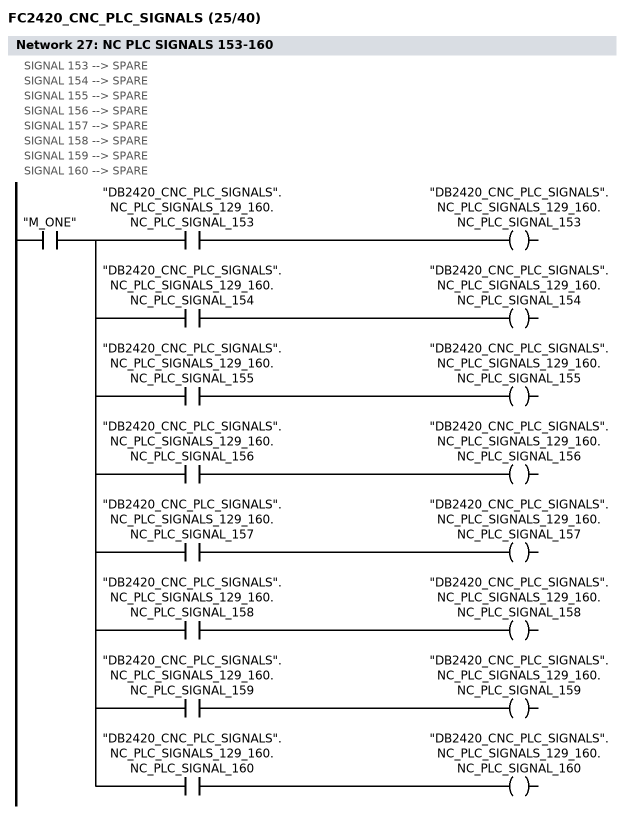
   RUNG wire#powerrail
      Contact( "M_ONE" )
      wire#w1
      Contact( "DB2420_CNC_PLC_SIGNALS".NC_PLC_SIGNALS_129_160.NC_PLC_SIGNAL_153 )
      Coil( "DB2420_CNC_PLC_SIGNALS".NC_PLC_SIGNALS_129_160.NC_PLC_SIGNAL_153 )
   END_RUNG
   RUNG wire#w1
      Contact( "DB2420_CNC_PLC_SIGNALS".NC_PLC_SIGNALS_129_160.NC_PLC_SIGNAL_154 )
      Coil( "DB2420_CNC_PLC_SIGNALS".NC_PLC_SIGNALS_129_160.NC_PLC_SIGNAL_154 )
   END_RUNG
   RUNG wire#w1
      Contact( "DB2420_CNC_PLC_SIGNALS".NC_PLC_SIGNALS_129_160.NC_PLC_SIGNAL_155 )
      Coil( "DB2420_CNC_PLC_SIGNALS".NC_PLC_SIGNALS_129_160.NC_PLC_SIGNAL_155 )
   END_RUNG
   RUNG wire#w1
      Contact( "DB2420_CNC_PLC_SIGNALS".NC_PLC_SIGNALS_129_160.NC_PLC_SIGNAL_156 )
      Coil( "DB2420_CNC_PLC_SIGNALS".NC_PLC_SIGNALS_129_160.NC_PLC_SIGNAL_156 )
   END_RUNG
   RUNG wire#w1
      Contact( "DB2420_CNC_PLC_SIGNALS".NC_PLC_SIGNALS_129_160.NC_PLC_SIGNAL_157 )
      Coil( "DB2420_CNC_PLC_SIGNALS".NC_PLC_SIGNALS_129_160.NC_PLC_SIGNAL_157 )
   END_RUNG
   RUNG wire#w1
      Contact( "DB2420_CNC_PLC_SIGNALS".NC_PLC_SIGNALS_129_160.NC_PLC_SIGNAL_158 )
      Coil( "DB2420_CNC_PLC_SIGNALS".NC_PLC_SIGNALS_129_160.NC_PLC_SIGNAL_158 )
   END_RUNG
   RUNG wire#w1
      Contact( "DB2420_CNC_PLC_SIGNALS".NC_PLC_SIGNALS_129_160.NC_PLC_SIGNAL_159 )
      Coil( "DB2420_CNC_PLC_SIGNALS".NC_PLC_SIGNALS_129_160.NC_PLC_SIGNAL_159 )
   END_RUNG
   RUNG wire#w1
      Contact( "DB2420_CNC_PLC_SIGNALS".NC_PLC_SIGNALS_129_160.NC_PLC_SIGNAL_160 )
      Coil( "DB2420_CNC_PLC_SIGNALS".NC_PLC_SIGNALS_129_160.NC_PLC_SIGNAL_160 )
   END_RUNG
   // the same network as SCL:
   "DB2420_CNC_PLC_SIGNALS".NC_PLC_SIGNALS_129_160.NC_PLC_SIGNAL_153 := "M_ONE" AND "DB2420_CNC_PLC_SIGNALS".NC_PLC_SIGNALS_129_160.NC_PLC_SIGNAL_153;
   "DB2420_CNC_PLC_SIGNALS".NC_PLC_SIGNALS_129_160.NC_PLC_SIGNAL_154 := "M_ONE" AND "DB2420_CNC_PLC_SIGNALS".NC_PLC_SIGNALS_129_160.NC_PLC_SIGNAL_154;
   "DB2420_CNC_PLC_SIGNALS".NC_PLC_SIGNALS_129_160.NC_PLC_SIGNAL_155 := "M_ONE" AND "DB2420_CNC_PLC_SIGNALS".NC_PLC_SIGNALS_129_160.NC_PLC_SIGNAL_155;
   "DB2420_CNC_PLC_SIGNALS".NC_PLC_SIGNALS_129_160.NC_PLC_SIGNAL_156 := "M_ONE" AND "DB2420_CNC_PLC_SIGNALS".NC_PLC_SIGNALS_129_160.NC_PLC_SIGNAL_156;
   "DB2420_CNC_PLC_SIGNALS".NC_PLC_SIGNALS_129_160.NC_PLC_SIGNAL_157 := "M_ONE" AND "DB2420_CNC_PLC_SIGNALS".NC_PLC_SIGNALS_129_160.NC_PLC_SIGNAL_157;
   "DB2420_CNC_PLC_SIGNALS".NC_PLC_SIGNALS_129_160.NC_PLC_SIGNAL_158 := "M_ONE" AND "DB2420_CNC_PLC_SIGNALS".NC_PLC_SIGNALS_129_160.NC_PLC_SIGNAL_158;
   "DB2420_CNC_PLC_SIGNALS".NC_PLC_SIGNALS_129_160.NC_PLC_SIGNAL_159 := "M_ONE" AND "DB2420_CNC_PLC_SIGNALS".NC_PLC_SIGNALS_129_160.NC_PLC_SIGNAL_159;
   "DB2420_CNC_PLC_SIGNALS".NC_PLC_SIGNALS_129_160.NC_PLC_SIGNAL_160 := "M_ONE" AND "DB2420_CNC_PLC_SIGNALS".NC_PLC_SIGNALS_129_160.NC_PLC_SIGNAL_160;
END_REGION

REGION Network 28: CALL FC21 NC PLC SIGNALS- $A_DBD[4060] / WRITE UNIT CYCLE SELECTION TO CNC
   // $A_DBD[1000] IN CNC
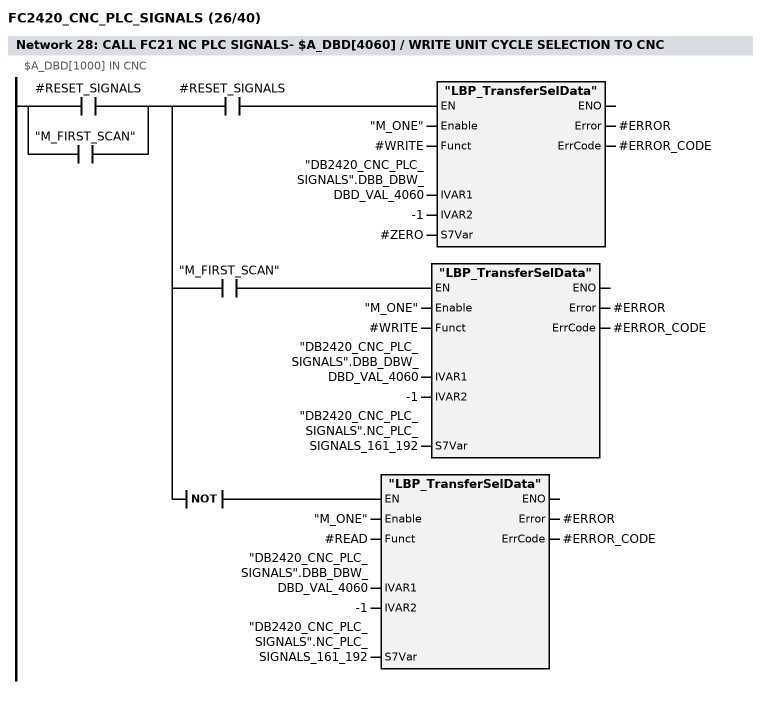
   RUNG wire#powerrail
      Contact( #RESET_SIGNALS )
      wire#w1
      Contact( #RESET_SIGNALS )
      "LBP_TransferSelData"(Enable := "M_ONE", Funct := #WRITE, IVAR1 := "DB2420_CNC_PLC_SIGNALS".DBB_DBW_DBD_VAL_4060, IVAR2 := -1, S7Var := #ZERO, Error => #ERROR, ErrCode => #ERROR_CODE)
   END_RUNG
   RUNG wire#powerrail
      Contact( "M_FIRST_SCAN" )
   END_RUNG wire#w1
   RUNG wire#w1
      Contact( "M_FIRST_SCAN" )
      "LBP_TransferSelData"(Enable := "M_ONE", Funct := #WRITE, IVAR1 := "DB2420_CNC_PLC_SIGNALS".DBB_DBW_DBD_VAL_4060, IVAR2 := -1, S7Var := "DB2420_CNC_PLC_SIGNALS".NC_PLC_SIGNALS_161_192, Error => #ERROR, ErrCode => #ERROR_CODE)
   END_RUNG
   RUNG wire#w1
      Not()
      "LBP_TransferSelData"(Enable := "M_ONE", Funct := #READ, IVAR1 := "DB2420_CNC_PLC_SIGNALS".DBB_DBW_DBD_VAL_4060, IVAR2 := -1, S7Var := "DB2420_CNC_PLC_SIGNALS".NC_PLC_SIGNALS_161_192, Error => #ERROR, ErrCode => #ERROR_CODE)
   END_RUNG
   // the same network as SCL:
   #_w1 := #RESET_SIGNALS OR "M_FIRST_SCAN";
   IF #_w1 AND #RESET_SIGNALS THEN
       "LBP_TransferSelData"(Enable := "M_ONE",
                             Funct := #WRITE,
                             IVAR1 := "DB2420_CNC_PLC_SIGNALS".DBB_DBW_DBD_VAL_4060,
                             IVAR2 := -1,
                             S7Var := #ZERO,
                             Error => #ERROR,
                             ErrCode => #ERROR_CODE);
   END_IF;
   IF #_w1 AND "M_FIRST_SCAN" THEN
       "LBP_TransferSelData"(Enable := "M_ONE",
                             Funct := #WRITE,
                             IVAR1 := "DB2420_CNC_PLC_SIGNALS".DBB_DBW_DBD_VAL_4060,
                             IVAR2 := -1,
                             S7Var := "DB2420_CNC_PLC_SIGNALS".NC_PLC_SIGNALS_161_192,
                             Error => #ERROR,
                             ErrCode => #ERROR_CODE);
   END_IF;
   IF NOT #_w1 THEN
       "LBP_TransferSelData"(Enable := "M_ONE",
                             Funct := #READ,
                             IVAR1 := "DB2420_CNC_PLC_SIGNALS".DBB_DBW_DBD_VAL_4060,
                             IVAR2 := -1,
                             S7Var := "DB2420_CNC_PLC_SIGNALS".NC_PLC_SIGNALS_161_192,
                             Error => #ERROR,
                             ErrCode => #ERROR_CODE);
   END_IF;
END_REGION

REGION Network 29: NC PLC SIGNALS 161-168
   // SIGNAL 161 --> SPARE
   // SIGNAL 162 --> SPARE
   // SIGNAL 163 --> SPARE
   // SIGNAL 164 --> SPARE
   // SIGNAL 165 --> SPARE
   // SIGNAL 166 --> SPARE
   // SIGNAL 167 --> SPARE
   // SIGNAL 168 --> SPARE
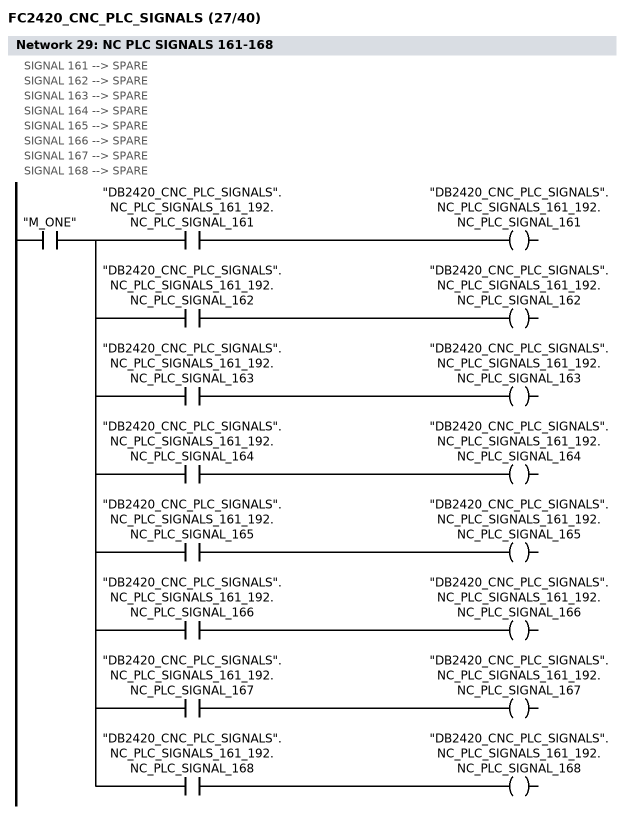
   RUNG wire#powerrail
      Contact( "M_ONE" )
      wire#w1
      Contact( "DB2420_CNC_PLC_SIGNALS".NC_PLC_SIGNALS_161_192.NC_PLC_SIGNAL_161 )
      Coil( "DB2420_CNC_PLC_SIGNALS".NC_PLC_SIGNALS_161_192.NC_PLC_SIGNAL_161 )
   END_RUNG
   RUNG wire#w1
      Contact( "DB2420_CNC_PLC_SIGNALS".NC_PLC_SIGNALS_161_192.NC_PLC_SIGNAL_162 )
      Coil( "DB2420_CNC_PLC_SIGNALS".NC_PLC_SIGNALS_161_192.NC_PLC_SIGNAL_162 )
   END_RUNG
   RUNG wire#w1
      Contact( "DB2420_CNC_PLC_SIGNALS".NC_PLC_SIGNALS_161_192.NC_PLC_SIGNAL_163 )
      Coil( "DB2420_CNC_PLC_SIGNALS".NC_PLC_SIGNALS_161_192.NC_PLC_SIGNAL_163 )
   END_RUNG
   RUNG wire#w1
      Contact( "DB2420_CNC_PLC_SIGNALS".NC_PLC_SIGNALS_161_192.NC_PLC_SIGNAL_164 )
      Coil( "DB2420_CNC_PLC_SIGNALS".NC_PLC_SIGNALS_161_192.NC_PLC_SIGNAL_164 )
   END_RUNG
   RUNG wire#w1
      Contact( "DB2420_CNC_PLC_SIGNALS".NC_PLC_SIGNALS_161_192.NC_PLC_SIGNAL_165 )
      Coil( "DB2420_CNC_PLC_SIGNALS".NC_PLC_SIGNALS_161_192.NC_PLC_SIGNAL_165 )
   END_RUNG
   RUNG wire#w1
      Contact( "DB2420_CNC_PLC_SIGNALS".NC_PLC_SIGNALS_161_192.NC_PLC_SIGNAL_166 )
      Coil( "DB2420_CNC_PLC_SIGNALS".NC_PLC_SIGNALS_161_192.NC_PLC_SIGNAL_166 )
   END_RUNG
   RUNG wire#w1
      Contact( "DB2420_CNC_PLC_SIGNALS".NC_PLC_SIGNALS_161_192.NC_PLC_SIGNAL_167 )
      Coil( "DB2420_CNC_PLC_SIGNALS".NC_PLC_SIGNALS_161_192.NC_PLC_SIGNAL_167 )
   END_RUNG
   RUNG wire#w1
      Contact( "DB2420_CNC_PLC_SIGNALS".NC_PLC_SIGNALS_161_192.NC_PLC_SIGNAL_168 )
      Coil( "DB2420_CNC_PLC_SIGNALS".NC_PLC_SIGNALS_161_192.NC_PLC_SIGNAL_168 )
   END_RUNG
   // the same network as SCL:
   "DB2420_CNC_PLC_SIGNALS".NC_PLC_SIGNALS_161_192.NC_PLC_SIGNAL_161 := "M_ONE" AND "DB2420_CNC_PLC_SIGNALS".NC_PLC_SIGNALS_161_192.NC_PLC_SIGNAL_161;
   "DB2420_CNC_PLC_SIGNALS".NC_PLC_SIGNALS_161_192.NC_PLC_SIGNAL_162 := "M_ONE" AND "DB2420_CNC_PLC_SIGNALS".NC_PLC_SIGNALS_161_192.NC_PLC_SIGNAL_162;
   "DB2420_CNC_PLC_SIGNALS".NC_PLC_SIGNALS_161_192.NC_PLC_SIGNAL_163 := "M_ONE" AND "DB2420_CNC_PLC_SIGNALS".NC_PLC_SIGNALS_161_192.NC_PLC_SIGNAL_163;
   "DB2420_CNC_PLC_SIGNALS".NC_PLC_SIGNALS_161_192.NC_PLC_SIGNAL_164 := "M_ONE" AND "DB2420_CNC_PLC_SIGNALS".NC_PLC_SIGNALS_161_192.NC_PLC_SIGNAL_164;
   "DB2420_CNC_PLC_SIGNALS".NC_PLC_SIGNALS_161_192.NC_PLC_SIGNAL_165 := "M_ONE" AND "DB2420_CNC_PLC_SIGNALS".NC_PLC_SIGNALS_161_192.NC_PLC_SIGNAL_165;
   "DB2420_CNC_PLC_SIGNALS".NC_PLC_SIGNALS_161_192.NC_PLC_SIGNAL_166 := "M_ONE" AND "DB2420_CNC_PLC_SIGNALS".NC_PLC_SIGNALS_161_192.NC_PLC_SIGNAL_166;
   "DB2420_CNC_PLC_SIGNALS".NC_PLC_SIGNALS_161_192.NC_PLC_SIGNAL_167 := "M_ONE" AND "DB2420_CNC_PLC_SIGNALS".NC_PLC_SIGNALS_161_192.NC_PLC_SIGNAL_167;
   "DB2420_CNC_PLC_SIGNALS".NC_PLC_SIGNALS_161_192.NC_PLC_SIGNAL_168 := "M_ONE" AND "DB2420_CNC_PLC_SIGNALS".NC_PLC_SIGNALS_161_192.NC_PLC_SIGNAL_168;
END_REGION

REGION Network 30: NC PLC SIGNALS 169-176
   // SIGNAL 169 --> SPARE
   // SIGNAL 170 --> SPARE
   // SIGNAL 171 --> SPARE
   // SIGNAL 172 --> SPARE
   // SIGNAL 173 --> SPARE
   // SIGNAL 174 --> SPARE
   // SIGNAL 175 --> SPARE
   // SIGNAL 176 --> SPARE
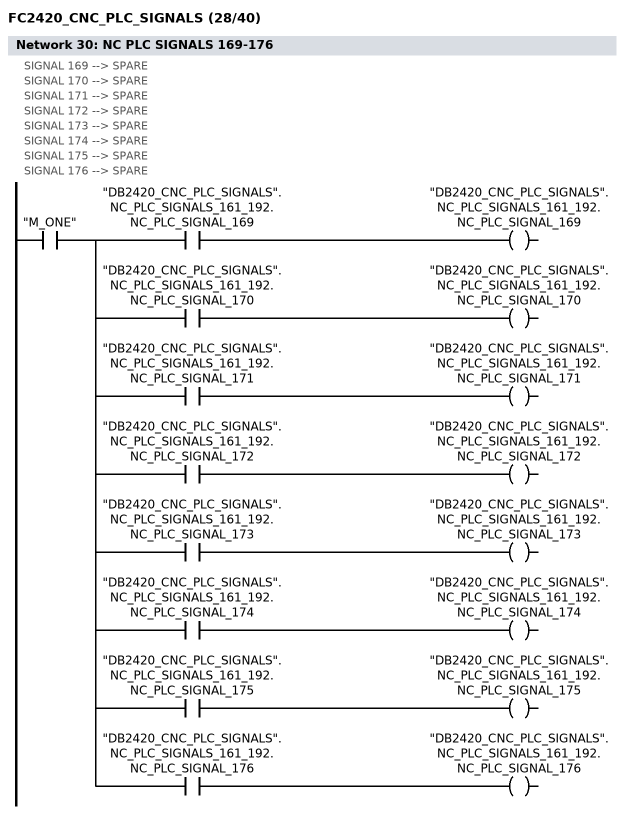
   RUNG wire#powerrail
      Contact( "M_ONE" )
      wire#w1
      Contact( "DB2420_CNC_PLC_SIGNALS".NC_PLC_SIGNALS_161_192.NC_PLC_SIGNAL_169 )
      Coil( "DB2420_CNC_PLC_SIGNALS".NC_PLC_SIGNALS_161_192.NC_PLC_SIGNAL_169 )
   END_RUNG
   RUNG wire#w1
      Contact( "DB2420_CNC_PLC_SIGNALS".NC_PLC_SIGNALS_161_192.NC_PLC_SIGNAL_170 )
      Coil( "DB2420_CNC_PLC_SIGNALS".NC_PLC_SIGNALS_161_192.NC_PLC_SIGNAL_170 )
   END_RUNG
   RUNG wire#w1
      Contact( "DB2420_CNC_PLC_SIGNALS".NC_PLC_SIGNALS_161_192.NC_PLC_SIGNAL_171 )
      Coil( "DB2420_CNC_PLC_SIGNALS".NC_PLC_SIGNALS_161_192.NC_PLC_SIGNAL_171 )
   END_RUNG
   RUNG wire#w1
      Contact( "DB2420_CNC_PLC_SIGNALS".NC_PLC_SIGNALS_161_192.NC_PLC_SIGNAL_172 )
      Coil( "DB2420_CNC_PLC_SIGNALS".NC_PLC_SIGNALS_161_192.NC_PLC_SIGNAL_172 )
   END_RUNG
   RUNG wire#w1
      Contact( "DB2420_CNC_PLC_SIGNALS".NC_PLC_SIGNALS_161_192.NC_PLC_SIGNAL_173 )
      Coil( "DB2420_CNC_PLC_SIGNALS".NC_PLC_SIGNALS_161_192.NC_PLC_SIGNAL_173 )
   END_RUNG
   RUNG wire#w1
      Contact( "DB2420_CNC_PLC_SIGNALS".NC_PLC_SIGNALS_161_192.NC_PLC_SIGNAL_174 )
      Coil( "DB2420_CNC_PLC_SIGNALS".NC_PLC_SIGNALS_161_192.NC_PLC_SIGNAL_174 )
   END_RUNG
   RUNG wire#w1
      Contact( "DB2420_CNC_PLC_SIGNALS".NC_PLC_SIGNALS_161_192.NC_PLC_SIGNAL_175 )
      Coil( "DB2420_CNC_PLC_SIGNALS".NC_PLC_SIGNALS_161_192.NC_PLC_SIGNAL_175 )
   END_RUNG
   RUNG wire#w1
      Contact( "DB2420_CNC_PLC_SIGNALS".NC_PLC_SIGNALS_161_192.NC_PLC_SIGNAL_176 )
      Coil( "DB2420_CNC_PLC_SIGNALS".NC_PLC_SIGNALS_161_192.NC_PLC_SIGNAL_176 )
   END_RUNG
   // the same network as SCL:
   "DB2420_CNC_PLC_SIGNALS".NC_PLC_SIGNALS_161_192.NC_PLC_SIGNAL_169 := "M_ONE" AND "DB2420_CNC_PLC_SIGNALS".NC_PLC_SIGNALS_161_192.NC_PLC_SIGNAL_169;
   "DB2420_CNC_PLC_SIGNALS".NC_PLC_SIGNALS_161_192.NC_PLC_SIGNAL_170 := "M_ONE" AND "DB2420_CNC_PLC_SIGNALS".NC_PLC_SIGNALS_161_192.NC_PLC_SIGNAL_170;
   "DB2420_CNC_PLC_SIGNALS".NC_PLC_SIGNALS_161_192.NC_PLC_SIGNAL_171 := "M_ONE" AND "DB2420_CNC_PLC_SIGNALS".NC_PLC_SIGNALS_161_192.NC_PLC_SIGNAL_171;
   "DB2420_CNC_PLC_SIGNALS".NC_PLC_SIGNALS_161_192.NC_PLC_SIGNAL_172 := "M_ONE" AND "DB2420_CNC_PLC_SIGNALS".NC_PLC_SIGNALS_161_192.NC_PLC_SIGNAL_172;
   "DB2420_CNC_PLC_SIGNALS".NC_PLC_SIGNALS_161_192.NC_PLC_SIGNAL_173 := "M_ONE" AND "DB2420_CNC_PLC_SIGNALS".NC_PLC_SIGNALS_161_192.NC_PLC_SIGNAL_173;
   "DB2420_CNC_PLC_SIGNALS".NC_PLC_SIGNALS_161_192.NC_PLC_SIGNAL_174 := "M_ONE" AND "DB2420_CNC_PLC_SIGNALS".NC_PLC_SIGNALS_161_192.NC_PLC_SIGNAL_174;
   "DB2420_CNC_PLC_SIGNALS".NC_PLC_SIGNALS_161_192.NC_PLC_SIGNAL_175 := "M_ONE" AND "DB2420_CNC_PLC_SIGNALS".NC_PLC_SIGNALS_161_192.NC_PLC_SIGNAL_175;
   "DB2420_CNC_PLC_SIGNALS".NC_PLC_SIGNALS_161_192.NC_PLC_SIGNAL_176 := "M_ONE" AND "DB2420_CNC_PLC_SIGNALS".NC_PLC_SIGNALS_161_192.NC_PLC_SIGNAL_176;
END_REGION

REGION Network 31: NC PLC SIGNALS 177-184
   // SIGNAL 177 --> SPARE
   // SIGNAL 178 --> SPARE
   // SIGNAL 179 --> SPARE
   // SIGNAL 180 --> SPARE
   // SIGNAL 181 --> SPARE
   // SIGNAL 182 --> SPARE
   // SIGNAL 183 --> SPARE
   // SIGNAL 184 --> SPARE
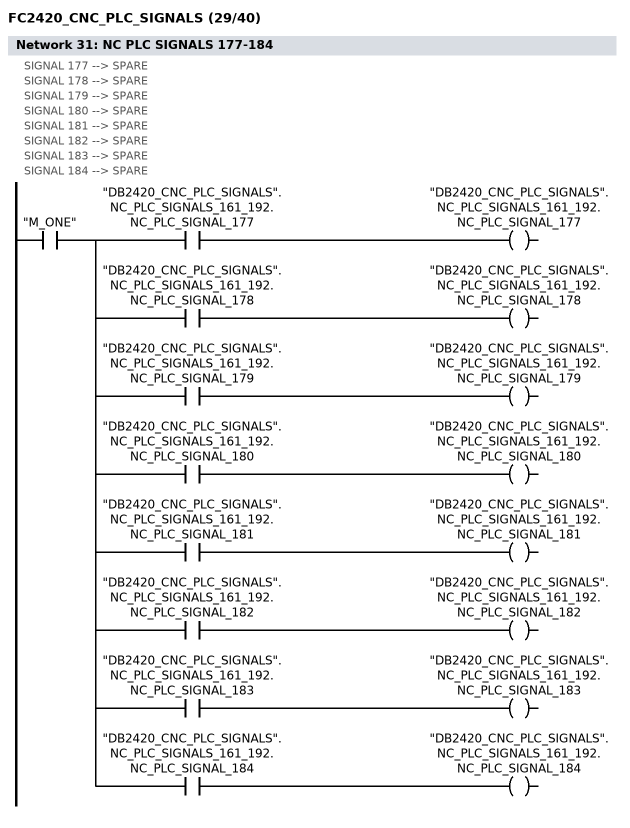
   RUNG wire#powerrail
      Contact( "M_ONE" )
      wire#w1
      Contact( "DB2420_CNC_PLC_SIGNALS".NC_PLC_SIGNALS_161_192.NC_PLC_SIGNAL_177 )
      Coil( "DB2420_CNC_PLC_SIGNALS".NC_PLC_SIGNALS_161_192.NC_PLC_SIGNAL_177 )
   END_RUNG
   RUNG wire#w1
      Contact( "DB2420_CNC_PLC_SIGNALS".NC_PLC_SIGNALS_161_192.NC_PLC_SIGNAL_178 )
      Coil( "DB2420_CNC_PLC_SIGNALS".NC_PLC_SIGNALS_161_192.NC_PLC_SIGNAL_178 )
   END_RUNG
   RUNG wire#w1
      Contact( "DB2420_CNC_PLC_SIGNALS".NC_PLC_SIGNALS_161_192.NC_PLC_SIGNAL_179 )
      Coil( "DB2420_CNC_PLC_SIGNALS".NC_PLC_SIGNALS_161_192.NC_PLC_SIGNAL_179 )
   END_RUNG
   RUNG wire#w1
      Contact( "DB2420_CNC_PLC_SIGNALS".NC_PLC_SIGNALS_161_192.NC_PLC_SIGNAL_180 )
      Coil( "DB2420_CNC_PLC_SIGNALS".NC_PLC_SIGNALS_161_192.NC_PLC_SIGNAL_180 )
   END_RUNG
   RUNG wire#w1
      Contact( "DB2420_CNC_PLC_SIGNALS".NC_PLC_SIGNALS_161_192.NC_PLC_SIGNAL_181 )
      Coil( "DB2420_CNC_PLC_SIGNALS".NC_PLC_SIGNALS_161_192.NC_PLC_SIGNAL_181 )
   END_RUNG
   RUNG wire#w1
      Contact( "DB2420_CNC_PLC_SIGNALS".NC_PLC_SIGNALS_161_192.NC_PLC_SIGNAL_182 )
      Coil( "DB2420_CNC_PLC_SIGNALS".NC_PLC_SIGNALS_161_192.NC_PLC_SIGNAL_182 )
   END_RUNG
   RUNG wire#w1
      Contact( "DB2420_CNC_PLC_SIGNALS".NC_PLC_SIGNALS_161_192.NC_PLC_SIGNAL_183 )
      Coil( "DB2420_CNC_PLC_SIGNALS".NC_PLC_SIGNALS_161_192.NC_PLC_SIGNAL_183 )
   END_RUNG
   RUNG wire#w1
      Contact( "DB2420_CNC_PLC_SIGNALS".NC_PLC_SIGNALS_161_192.NC_PLC_SIGNAL_184 )
      Coil( "DB2420_CNC_PLC_SIGNALS".NC_PLC_SIGNALS_161_192.NC_PLC_SIGNAL_184 )
   END_RUNG
   // the same network as SCL:
   "DB2420_CNC_PLC_SIGNALS".NC_PLC_SIGNALS_161_192.NC_PLC_SIGNAL_177 := "M_ONE" AND "DB2420_CNC_PLC_SIGNALS".NC_PLC_SIGNALS_161_192.NC_PLC_SIGNAL_177;
   "DB2420_CNC_PLC_SIGNALS".NC_PLC_SIGNALS_161_192.NC_PLC_SIGNAL_178 := "M_ONE" AND "DB2420_CNC_PLC_SIGNALS".NC_PLC_SIGNALS_161_192.NC_PLC_SIGNAL_178;
   "DB2420_CNC_PLC_SIGNALS".NC_PLC_SIGNALS_161_192.NC_PLC_SIGNAL_179 := "M_ONE" AND "DB2420_CNC_PLC_SIGNALS".NC_PLC_SIGNALS_161_192.NC_PLC_SIGNAL_179;
   "DB2420_CNC_PLC_SIGNALS".NC_PLC_SIGNALS_161_192.NC_PLC_SIGNAL_180 := "M_ONE" AND "DB2420_CNC_PLC_SIGNALS".NC_PLC_SIGNALS_161_192.NC_PLC_SIGNAL_180;
   "DB2420_CNC_PLC_SIGNALS".NC_PLC_SIGNALS_161_192.NC_PLC_SIGNAL_181 := "M_ONE" AND "DB2420_CNC_PLC_SIGNALS".NC_PLC_SIGNALS_161_192.NC_PLC_SIGNAL_181;
   "DB2420_CNC_PLC_SIGNALS".NC_PLC_SIGNALS_161_192.NC_PLC_SIGNAL_182 := "M_ONE" AND "DB2420_CNC_PLC_SIGNALS".NC_PLC_SIGNALS_161_192.NC_PLC_SIGNAL_182;
   "DB2420_CNC_PLC_SIGNALS".NC_PLC_SIGNALS_161_192.NC_PLC_SIGNAL_183 := "M_ONE" AND "DB2420_CNC_PLC_SIGNALS".NC_PLC_SIGNALS_161_192.NC_PLC_SIGNAL_183;
   "DB2420_CNC_PLC_SIGNALS".NC_PLC_SIGNALS_161_192.NC_PLC_SIGNAL_184 := "M_ONE" AND "DB2420_CNC_PLC_SIGNALS".NC_PLC_SIGNALS_161_192.NC_PLC_SIGNAL_184;
END_REGION

REGION Network 32: NC PLC SIGNALS 185-192
   // SIGNAL 185 --> SPARE
   // SIGNAL 186 --> SPARE
   // SIGNAL 187 --> SPARE
   // SIGNAL 188 --> SPARE
   // SIGNAL 189 --> SPARE
   // SIGNAL 190 --> SPARE
   // SIGNAL 191 --> SPARE
   // SIGNAL 192 --> SPARE
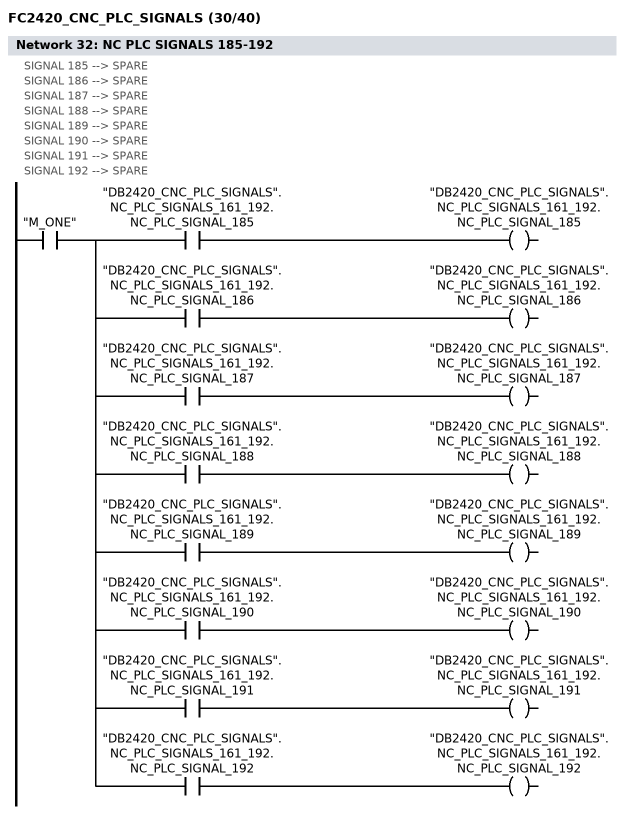
   RUNG wire#powerrail
      Contact( "M_ONE" )
      wire#w1
      Contact( "DB2420_CNC_PLC_SIGNALS".NC_PLC_SIGNALS_161_192.NC_PLC_SIGNAL_185 )
      Coil( "DB2420_CNC_PLC_SIGNALS".NC_PLC_SIGNALS_161_192.NC_PLC_SIGNAL_185 )
   END_RUNG
   RUNG wire#w1
      Contact( "DB2420_CNC_PLC_SIGNALS".NC_PLC_SIGNALS_161_192.NC_PLC_SIGNAL_186 )
      Coil( "DB2420_CNC_PLC_SIGNALS".NC_PLC_SIGNALS_161_192.NC_PLC_SIGNAL_186 )
   END_RUNG
   RUNG wire#w1
      Contact( "DB2420_CNC_PLC_SIGNALS".NC_PLC_SIGNALS_161_192.NC_PLC_SIGNAL_187 )
      Coil( "DB2420_CNC_PLC_SIGNALS".NC_PLC_SIGNALS_161_192.NC_PLC_SIGNAL_187 )
   END_RUNG
   RUNG wire#w1
      Contact( "DB2420_CNC_PLC_SIGNALS".NC_PLC_SIGNALS_161_192.NC_PLC_SIGNAL_188 )
      Coil( "DB2420_CNC_PLC_SIGNALS".NC_PLC_SIGNALS_161_192.NC_PLC_SIGNAL_188 )
   END_RUNG
   RUNG wire#w1
      Contact( "DB2420_CNC_PLC_SIGNALS".NC_PLC_SIGNALS_161_192.NC_PLC_SIGNAL_189 )
      Coil( "DB2420_CNC_PLC_SIGNALS".NC_PLC_SIGNALS_161_192.NC_PLC_SIGNAL_189 )
   END_RUNG
   RUNG wire#w1
      Contact( "DB2420_CNC_PLC_SIGNALS".NC_PLC_SIGNALS_161_192.NC_PLC_SIGNAL_190 )
      Coil( "DB2420_CNC_PLC_SIGNALS".NC_PLC_SIGNALS_161_192.NC_PLC_SIGNAL_190 )
   END_RUNG
   RUNG wire#w1
      Contact( "DB2420_CNC_PLC_SIGNALS".NC_PLC_SIGNALS_161_192.NC_PLC_SIGNAL_191 )
      Coil( "DB2420_CNC_PLC_SIGNALS".NC_PLC_SIGNALS_161_192.NC_PLC_SIGNAL_191 )
   END_RUNG
   RUNG wire#w1
      Contact( "DB2420_CNC_PLC_SIGNALS".NC_PLC_SIGNALS_161_192.NC_PLC_SIGNAL_192 )
      Coil( "DB2420_CNC_PLC_SIGNALS".NC_PLC_SIGNALS_161_192.NC_PLC_SIGNAL_192 )
   END_RUNG
   // the same network as SCL:
   "DB2420_CNC_PLC_SIGNALS".NC_PLC_SIGNALS_161_192.NC_PLC_SIGNAL_185 := "M_ONE" AND "DB2420_CNC_PLC_SIGNALS".NC_PLC_SIGNALS_161_192.NC_PLC_SIGNAL_185;
   "DB2420_CNC_PLC_SIGNALS".NC_PLC_SIGNALS_161_192.NC_PLC_SIGNAL_186 := "M_ONE" AND "DB2420_CNC_PLC_SIGNALS".NC_PLC_SIGNALS_161_192.NC_PLC_SIGNAL_186;
   "DB2420_CNC_PLC_SIGNALS".NC_PLC_SIGNALS_161_192.NC_PLC_SIGNAL_187 := "M_ONE" AND "DB2420_CNC_PLC_SIGNALS".NC_PLC_SIGNALS_161_192.NC_PLC_SIGNAL_187;
   "DB2420_CNC_PLC_SIGNALS".NC_PLC_SIGNALS_161_192.NC_PLC_SIGNAL_188 := "M_ONE" AND "DB2420_CNC_PLC_SIGNALS".NC_PLC_SIGNALS_161_192.NC_PLC_SIGNAL_188;
   "DB2420_CNC_PLC_SIGNALS".NC_PLC_SIGNALS_161_192.NC_PLC_SIGNAL_189 := "M_ONE" AND "DB2420_CNC_PLC_SIGNALS".NC_PLC_SIGNALS_161_192.NC_PLC_SIGNAL_189;
   "DB2420_CNC_PLC_SIGNALS".NC_PLC_SIGNALS_161_192.NC_PLC_SIGNAL_190 := "M_ONE" AND "DB2420_CNC_PLC_SIGNALS".NC_PLC_SIGNALS_161_192.NC_PLC_SIGNAL_190;
   "DB2420_CNC_PLC_SIGNALS".NC_PLC_SIGNALS_161_192.NC_PLC_SIGNAL_191 := "M_ONE" AND "DB2420_CNC_PLC_SIGNALS".NC_PLC_SIGNALS_161_192.NC_PLC_SIGNAL_191;
   "DB2420_CNC_PLC_SIGNALS".NC_PLC_SIGNALS_161_192.NC_PLC_SIGNAL_192 := "M_ONE" AND "DB2420_CNC_PLC_SIGNALS".NC_PLC_SIGNALS_161_192.NC_PLC_SIGNAL_192;
END_REGION

REGION Network 33: CALL FC21 NC PLC SIGNALS- $A_DBD[4064] / WRITE UNIT CYCLE SELECTION TO CNC
   // $A_DBD[1000] IN CNC
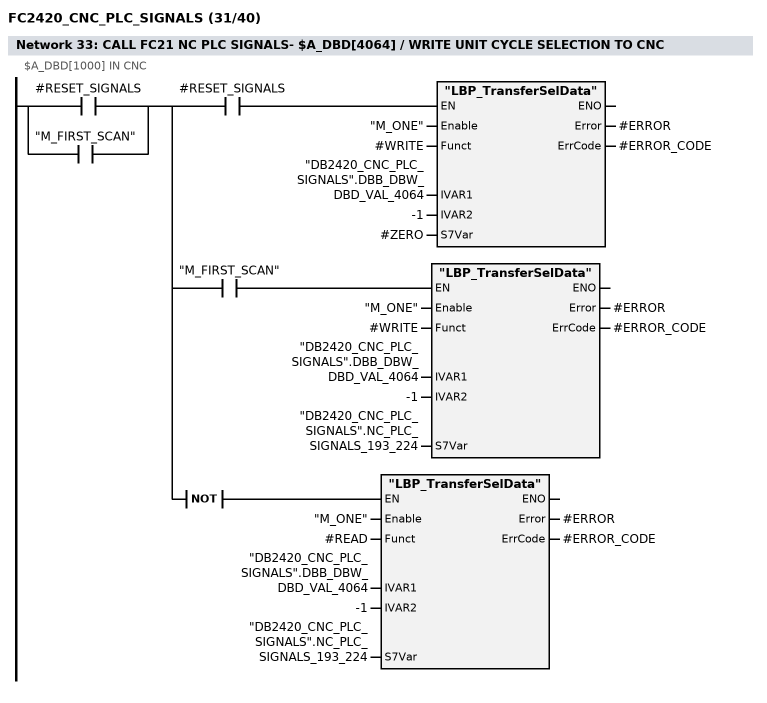
   RUNG wire#powerrail
      Contact( #RESET_SIGNALS )
      wire#w1
      Contact( #RESET_SIGNALS )
      "LBP_TransferSelData"(Enable := "M_ONE", Funct := #WRITE, IVAR1 := "DB2420_CNC_PLC_SIGNALS".DBB_DBW_DBD_VAL_4064, IVAR2 := -1, S7Var := #ZERO, Error => #ERROR, ErrCode => #ERROR_CODE)
   END_RUNG
   RUNG wire#powerrail
      Contact( "M_FIRST_SCAN" )
   END_RUNG wire#w1
   RUNG wire#w1
      Contact( "M_FIRST_SCAN" )
      "LBP_TransferSelData"(Enable := "M_ONE", Funct := #WRITE, IVAR1 := "DB2420_CNC_PLC_SIGNALS".DBB_DBW_DBD_VAL_4064, IVAR2 := -1, S7Var := "DB2420_CNC_PLC_SIGNALS".NC_PLC_SIGNALS_193_224, Error => #ERROR, ErrCode => #ERROR_CODE)
   END_RUNG
   RUNG wire#w1
      Not()
      "LBP_TransferSelData"(Enable := "M_ONE", Funct := #READ, IVAR1 := "DB2420_CNC_PLC_SIGNALS".DBB_DBW_DBD_VAL_4064, IVAR2 := -1, S7Var := "DB2420_CNC_PLC_SIGNALS".NC_PLC_SIGNALS_193_224, Error => #ERROR, ErrCode => #ERROR_CODE)
   END_RUNG
   // the same network as SCL:
   #_w1 := #RESET_SIGNALS OR "M_FIRST_SCAN";
   IF #_w1 AND #RESET_SIGNALS THEN
       "LBP_TransferSelData"(Enable := "M_ONE",
                             Funct := #WRITE,
                             IVAR1 := "DB2420_CNC_PLC_SIGNALS".DBB_DBW_DBD_VAL_4064,
                             IVAR2 := -1,
                             S7Var := #ZERO,
                             Error => #ERROR,
                             ErrCode => #ERROR_CODE);
   END_IF;
   IF #_w1 AND "M_FIRST_SCAN" THEN
       "LBP_TransferSelData"(Enable := "M_ONE",
                             Funct := #WRITE,
                             IVAR1 := "DB2420_CNC_PLC_SIGNALS".DBB_DBW_DBD_VAL_4064,
                             IVAR2 := -1,
                             S7Var := "DB2420_CNC_PLC_SIGNALS".NC_PLC_SIGNALS_193_224,
                             Error => #ERROR,
                             ErrCode => #ERROR_CODE);
   END_IF;
   IF NOT #_w1 THEN
       "LBP_TransferSelData"(Enable := "M_ONE",
                             Funct := #READ,
                             IVAR1 := "DB2420_CNC_PLC_SIGNALS".DBB_DBW_DBD_VAL_4064,
                             IVAR2 := -1,
                             S7Var := "DB2420_CNC_PLC_SIGNALS".NC_PLC_SIGNALS_193_224,
                             Error => #ERROR,
                             ErrCode => #ERROR_CODE);
   END_IF;
END_REGION

REGION Network 34: NC PLC SIGNALS 193-200
   // SIGNAL 193 --> SPARE
   // SIGNAL 194 --> SPARE
   // SIGNAL 195 --> SPARE
   // SIGNAL 196 --> SPARE
   // SIGNAL 197 --> SPARE
   // SIGNAL 198 --> SPARE
   // SIGNAL 199 --> SPARE
   // SIGNAL 200 --> SPARE
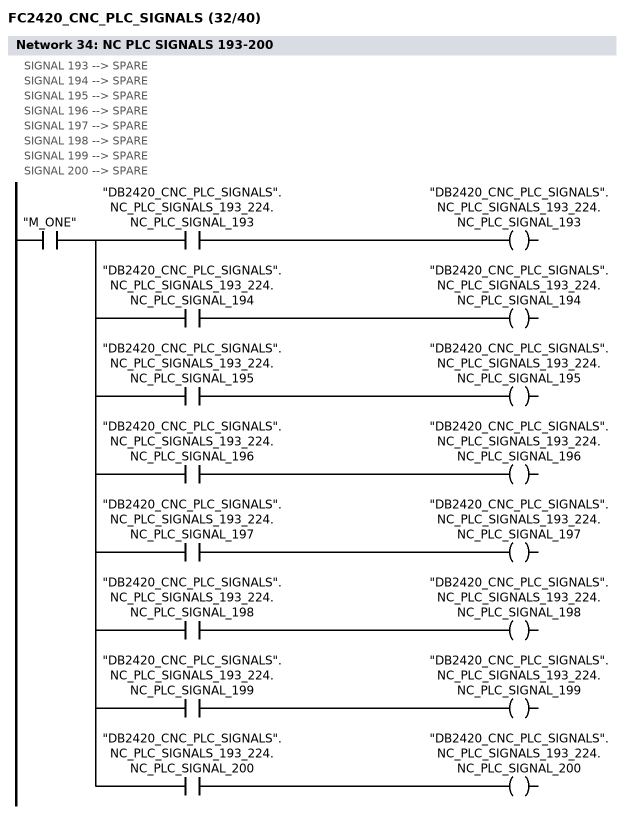
   RUNG wire#powerrail
      Contact( "M_ONE" )
      wire#w1
      Contact( "DB2420_CNC_PLC_SIGNALS".NC_PLC_SIGNALS_193_224.NC_PLC_SIGNAL_193 )
      Coil( "DB2420_CNC_PLC_SIGNALS".NC_PLC_SIGNALS_193_224.NC_PLC_SIGNAL_193 )
   END_RUNG
   RUNG wire#w1
      Contact( "DB2420_CNC_PLC_SIGNALS".NC_PLC_SIGNALS_193_224.NC_PLC_SIGNAL_194 )
      Coil( "DB2420_CNC_PLC_SIGNALS".NC_PLC_SIGNALS_193_224.NC_PLC_SIGNAL_194 )
   END_RUNG
   RUNG wire#w1
      Contact( "DB2420_CNC_PLC_SIGNALS".NC_PLC_SIGNALS_193_224.NC_PLC_SIGNAL_195 )
      Coil( "DB2420_CNC_PLC_SIGNALS".NC_PLC_SIGNALS_193_224.NC_PLC_SIGNAL_195 )
   END_RUNG
   RUNG wire#w1
      Contact( "DB2420_CNC_PLC_SIGNALS".NC_PLC_SIGNALS_193_224.NC_PLC_SIGNAL_196 )
      Coil( "DB2420_CNC_PLC_SIGNALS".NC_PLC_SIGNALS_193_224.NC_PLC_SIGNAL_196 )
   END_RUNG
   RUNG wire#w1
      Contact( "DB2420_CNC_PLC_SIGNALS".NC_PLC_SIGNALS_193_224.NC_PLC_SIGNAL_197 )
      Coil( "DB2420_CNC_PLC_SIGNALS".NC_PLC_SIGNALS_193_224.NC_PLC_SIGNAL_197 )
   END_RUNG
   RUNG wire#w1
      Contact( "DB2420_CNC_PLC_SIGNALS".NC_PLC_SIGNALS_193_224.NC_PLC_SIGNAL_198 )
      Coil( "DB2420_CNC_PLC_SIGNALS".NC_PLC_SIGNALS_193_224.NC_PLC_SIGNAL_198 )
   END_RUNG
   RUNG wire#w1
      Contact( "DB2420_CNC_PLC_SIGNALS".NC_PLC_SIGNALS_193_224.NC_PLC_SIGNAL_199 )
      Coil( "DB2420_CNC_PLC_SIGNALS".NC_PLC_SIGNALS_193_224.NC_PLC_SIGNAL_199 )
   END_RUNG
   RUNG wire#w1
      Contact( "DB2420_CNC_PLC_SIGNALS".NC_PLC_SIGNALS_193_224.NC_PLC_SIGNAL_200 )
      Coil( "DB2420_CNC_PLC_SIGNALS".NC_PLC_SIGNALS_193_224.NC_PLC_SIGNAL_200 )
   END_RUNG
   // the same network as SCL:
   "DB2420_CNC_PLC_SIGNALS".NC_PLC_SIGNALS_193_224.NC_PLC_SIGNAL_193 := "M_ONE" AND "DB2420_CNC_PLC_SIGNALS".NC_PLC_SIGNALS_193_224.NC_PLC_SIGNAL_193;
   "DB2420_CNC_PLC_SIGNALS".NC_PLC_SIGNALS_193_224.NC_PLC_SIGNAL_194 := "M_ONE" AND "DB2420_CNC_PLC_SIGNALS".NC_PLC_SIGNALS_193_224.NC_PLC_SIGNAL_194;
   "DB2420_CNC_PLC_SIGNALS".NC_PLC_SIGNALS_193_224.NC_PLC_SIGNAL_195 := "M_ONE" AND "DB2420_CNC_PLC_SIGNALS".NC_PLC_SIGNALS_193_224.NC_PLC_SIGNAL_195;
   "DB2420_CNC_PLC_SIGNALS".NC_PLC_SIGNALS_193_224.NC_PLC_SIGNAL_196 := "M_ONE" AND "DB2420_CNC_PLC_SIGNALS".NC_PLC_SIGNALS_193_224.NC_PLC_SIGNAL_196;
   "DB2420_CNC_PLC_SIGNALS".NC_PLC_SIGNALS_193_224.NC_PLC_SIGNAL_197 := "M_ONE" AND "DB2420_CNC_PLC_SIGNALS".NC_PLC_SIGNALS_193_224.NC_PLC_SIGNAL_197;
   "DB2420_CNC_PLC_SIGNALS".NC_PLC_SIGNALS_193_224.NC_PLC_SIGNAL_198 := "M_ONE" AND "DB2420_CNC_PLC_SIGNALS".NC_PLC_SIGNALS_193_224.NC_PLC_SIGNAL_198;
   "DB2420_CNC_PLC_SIGNALS".NC_PLC_SIGNALS_193_224.NC_PLC_SIGNAL_199 := "M_ONE" AND "DB2420_CNC_PLC_SIGNALS".NC_PLC_SIGNALS_193_224.NC_PLC_SIGNAL_199;
   "DB2420_CNC_PLC_SIGNALS".NC_PLC_SIGNALS_193_224.NC_PLC_SIGNAL_200 := "M_ONE" AND "DB2420_CNC_PLC_SIGNALS".NC_PLC_SIGNALS_193_224.NC_PLC_SIGNAL_200;
END_REGION

REGION Network 35: NC PLC SIGNALS 201-208
   // SIGNAL 201 --> SPARE
   // SIGNAL 202 --> SPARE
   // SIGNAL 203 --> SPARE
   // SIGNAL 204 --> SPARE
   // SIGNAL 205 --> SPARE
   // SIGNAL 206 --> SPARE
   // SIGNAL 207 --> SPARE
   // SIGNAL 208 --> SPARE
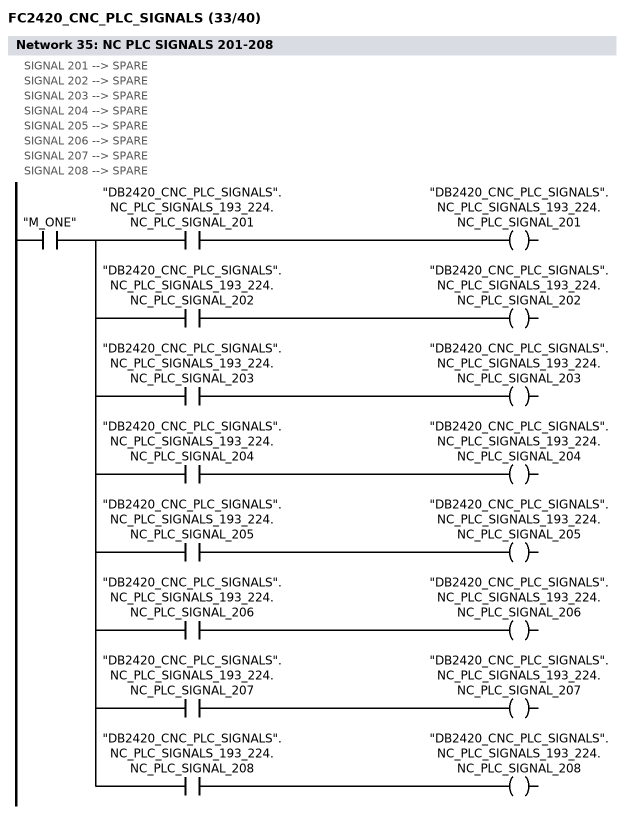
   RUNG wire#powerrail
      Contact( "M_ONE" )
      wire#w1
      Contact( "DB2420_CNC_PLC_SIGNALS".NC_PLC_SIGNALS_193_224.NC_PLC_SIGNAL_201 )
      Coil( "DB2420_CNC_PLC_SIGNALS".NC_PLC_SIGNALS_193_224.NC_PLC_SIGNAL_201 )
   END_RUNG
   RUNG wire#w1
      Contact( "DB2420_CNC_PLC_SIGNALS".NC_PLC_SIGNALS_193_224.NC_PLC_SIGNAL_202 )
      Coil( "DB2420_CNC_PLC_SIGNALS".NC_PLC_SIGNALS_193_224.NC_PLC_SIGNAL_202 )
   END_RUNG
   RUNG wire#w1
      Contact( "DB2420_CNC_PLC_SIGNALS".NC_PLC_SIGNALS_193_224.NC_PLC_SIGNAL_203 )
      Coil( "DB2420_CNC_PLC_SIGNALS".NC_PLC_SIGNALS_193_224.NC_PLC_SIGNAL_203 )
   END_RUNG
   RUNG wire#w1
      Contact( "DB2420_CNC_PLC_SIGNALS".NC_PLC_SIGNALS_193_224.NC_PLC_SIGNAL_204 )
      Coil( "DB2420_CNC_PLC_SIGNALS".NC_PLC_SIGNALS_193_224.NC_PLC_SIGNAL_204 )
   END_RUNG
   RUNG wire#w1
      Contact( "DB2420_CNC_PLC_SIGNALS".NC_PLC_SIGNALS_193_224.NC_PLC_SIGNAL_205 )
      Coil( "DB2420_CNC_PLC_SIGNALS".NC_PLC_SIGNALS_193_224.NC_PLC_SIGNAL_205 )
   END_RUNG
   RUNG wire#w1
      Contact( "DB2420_CNC_PLC_SIGNALS".NC_PLC_SIGNALS_193_224.NC_PLC_SIGNAL_206 )
      Coil( "DB2420_CNC_PLC_SIGNALS".NC_PLC_SIGNALS_193_224.NC_PLC_SIGNAL_206 )
   END_RUNG
   RUNG wire#w1
      Contact( "DB2420_CNC_PLC_SIGNALS".NC_PLC_SIGNALS_193_224.NC_PLC_SIGNAL_207 )
      Coil( "DB2420_CNC_PLC_SIGNALS".NC_PLC_SIGNALS_193_224.NC_PLC_SIGNAL_207 )
   END_RUNG
   RUNG wire#w1
      Contact( "DB2420_CNC_PLC_SIGNALS".NC_PLC_SIGNALS_193_224.NC_PLC_SIGNAL_208 )
      Coil( "DB2420_CNC_PLC_SIGNALS".NC_PLC_SIGNALS_193_224.NC_PLC_SIGNAL_208 )
   END_RUNG
   // the same network as SCL:
   "DB2420_CNC_PLC_SIGNALS".NC_PLC_SIGNALS_193_224.NC_PLC_SIGNAL_201 := "M_ONE" AND "DB2420_CNC_PLC_SIGNALS".NC_PLC_SIGNALS_193_224.NC_PLC_SIGNAL_201;
   "DB2420_CNC_PLC_SIGNALS".NC_PLC_SIGNALS_193_224.NC_PLC_SIGNAL_202 := "M_ONE" AND "DB2420_CNC_PLC_SIGNALS".NC_PLC_SIGNALS_193_224.NC_PLC_SIGNAL_202;
   "DB2420_CNC_PLC_SIGNALS".NC_PLC_SIGNALS_193_224.NC_PLC_SIGNAL_203 := "M_ONE" AND "DB2420_CNC_PLC_SIGNALS".NC_PLC_SIGNALS_193_224.NC_PLC_SIGNAL_203;
   "DB2420_CNC_PLC_SIGNALS".NC_PLC_SIGNALS_193_224.NC_PLC_SIGNAL_204 := "M_ONE" AND "DB2420_CNC_PLC_SIGNALS".NC_PLC_SIGNALS_193_224.NC_PLC_SIGNAL_204;
   "DB2420_CNC_PLC_SIGNALS".NC_PLC_SIGNALS_193_224.NC_PLC_SIGNAL_205 := "M_ONE" AND "DB2420_CNC_PLC_SIGNALS".NC_PLC_SIGNALS_193_224.NC_PLC_SIGNAL_205;
   "DB2420_CNC_PLC_SIGNALS".NC_PLC_SIGNALS_193_224.NC_PLC_SIGNAL_206 := "M_ONE" AND "DB2420_CNC_PLC_SIGNALS".NC_PLC_SIGNALS_193_224.NC_PLC_SIGNAL_206;
   "DB2420_CNC_PLC_SIGNALS".NC_PLC_SIGNALS_193_224.NC_PLC_SIGNAL_207 := "M_ONE" AND "DB2420_CNC_PLC_SIGNALS".NC_PLC_SIGNALS_193_224.NC_PLC_SIGNAL_207;
   "DB2420_CNC_PLC_SIGNALS".NC_PLC_SIGNALS_193_224.NC_PLC_SIGNAL_208 := "M_ONE" AND "DB2420_CNC_PLC_SIGNALS".NC_PLC_SIGNALS_193_224.NC_PLC_SIGNAL_208;
END_REGION

REGION Network 36: NC PLC SIGNALS 209-216
   // SIGNAL 209 --> SPARE
   // SIGNAL 210 --> SPARE
   // SIGNAL 211 --> SPARE
   // SIGNAL 212 --> SPARE
   // SIGNAL 213 --> SPARE
   // SIGNAL 214 --> SPARE
   // SIGNAL 215 --> SPARE
   // SIGNAL 216 --> SPARE
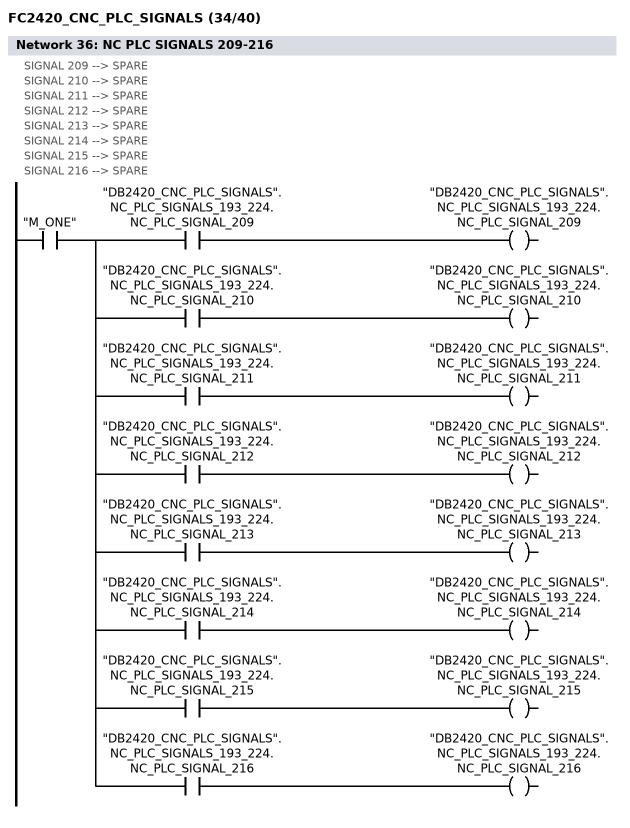
   RUNG wire#powerrail
      Contact( "M_ONE" )
      wire#w1
      Contact( "DB2420_CNC_PLC_SIGNALS".NC_PLC_SIGNALS_193_224.NC_PLC_SIGNAL_209 )
      Coil( "DB2420_CNC_PLC_SIGNALS".NC_PLC_SIGNALS_193_224.NC_PLC_SIGNAL_209 )
   END_RUNG
   RUNG wire#w1
      Contact( "DB2420_CNC_PLC_SIGNALS".NC_PLC_SIGNALS_193_224.NC_PLC_SIGNAL_210 )
      Coil( "DB2420_CNC_PLC_SIGNALS".NC_PLC_SIGNALS_193_224.NC_PLC_SIGNAL_210 )
   END_RUNG
   RUNG wire#w1
      Contact( "DB2420_CNC_PLC_SIGNALS".NC_PLC_SIGNALS_193_224.NC_PLC_SIGNAL_211 )
      Coil( "DB2420_CNC_PLC_SIGNALS".NC_PLC_SIGNALS_193_224.NC_PLC_SIGNAL_211 )
   END_RUNG
   RUNG wire#w1
      Contact( "DB2420_CNC_PLC_SIGNALS".NC_PLC_SIGNALS_193_224.NC_PLC_SIGNAL_212 )
      Coil( "DB2420_CNC_PLC_SIGNALS".NC_PLC_SIGNALS_193_224.NC_PLC_SIGNAL_212 )
   END_RUNG
   RUNG wire#w1
      Contact( "DB2420_CNC_PLC_SIGNALS".NC_PLC_SIGNALS_193_224.NC_PLC_SIGNAL_213 )
      Coil( "DB2420_CNC_PLC_SIGNALS".NC_PLC_SIGNALS_193_224.NC_PLC_SIGNAL_213 )
   END_RUNG
   RUNG wire#w1
      Contact( "DB2420_CNC_PLC_SIGNALS".NC_PLC_SIGNALS_193_224.NC_PLC_SIGNAL_214 )
      Coil( "DB2420_CNC_PLC_SIGNALS".NC_PLC_SIGNALS_193_224.NC_PLC_SIGNAL_214 )
   END_RUNG
   RUNG wire#w1
      Contact( "DB2420_CNC_PLC_SIGNALS".NC_PLC_SIGNALS_193_224.NC_PLC_SIGNAL_215 )
      Coil( "DB2420_CNC_PLC_SIGNALS".NC_PLC_SIGNALS_193_224.NC_PLC_SIGNAL_215 )
   END_RUNG
   RUNG wire#w1
      Contact( "DB2420_CNC_PLC_SIGNALS".NC_PLC_SIGNALS_193_224.NC_PLC_SIGNAL_216 )
      Coil( "DB2420_CNC_PLC_SIGNALS".NC_PLC_SIGNALS_193_224.NC_PLC_SIGNAL_216 )
   END_RUNG
   // the same network as SCL:
   "DB2420_CNC_PLC_SIGNALS".NC_PLC_SIGNALS_193_224.NC_PLC_SIGNAL_209 := "M_ONE" AND "DB2420_CNC_PLC_SIGNALS".NC_PLC_SIGNALS_193_224.NC_PLC_SIGNAL_209;
   "DB2420_CNC_PLC_SIGNALS".NC_PLC_SIGNALS_193_224.NC_PLC_SIGNAL_210 := "M_ONE" AND "DB2420_CNC_PLC_SIGNALS".NC_PLC_SIGNALS_193_224.NC_PLC_SIGNAL_210;
   "DB2420_CNC_PLC_SIGNALS".NC_PLC_SIGNALS_193_224.NC_PLC_SIGNAL_211 := "M_ONE" AND "DB2420_CNC_PLC_SIGNALS".NC_PLC_SIGNALS_193_224.NC_PLC_SIGNAL_211;
   "DB2420_CNC_PLC_SIGNALS".NC_PLC_SIGNALS_193_224.NC_PLC_SIGNAL_212 := "M_ONE" AND "DB2420_CNC_PLC_SIGNALS".NC_PLC_SIGNALS_193_224.NC_PLC_SIGNAL_212;
   "DB2420_CNC_PLC_SIGNALS".NC_PLC_SIGNALS_193_224.NC_PLC_SIGNAL_213 := "M_ONE" AND "DB2420_CNC_PLC_SIGNALS".NC_PLC_SIGNALS_193_224.NC_PLC_SIGNAL_213;
   "DB2420_CNC_PLC_SIGNALS".NC_PLC_SIGNALS_193_224.NC_PLC_SIGNAL_214 := "M_ONE" AND "DB2420_CNC_PLC_SIGNALS".NC_PLC_SIGNALS_193_224.NC_PLC_SIGNAL_214;
   "DB2420_CNC_PLC_SIGNALS".NC_PLC_SIGNALS_193_224.NC_PLC_SIGNAL_215 := "M_ONE" AND "DB2420_CNC_PLC_SIGNALS".NC_PLC_SIGNALS_193_224.NC_PLC_SIGNAL_215;
   "DB2420_CNC_PLC_SIGNALS".NC_PLC_SIGNALS_193_224.NC_PLC_SIGNAL_216 := "M_ONE" AND "DB2420_CNC_PLC_SIGNALS".NC_PLC_SIGNALS_193_224.NC_PLC_SIGNAL_216;
END_REGION

REGION Network 37: NC PLC SIGNALS 217-224
   // SIGNAL 217 --> SPARE
   // SIGNAL 218 --> SPARE
   // SIGNAL 219 --> SPARE
   // SIGNAL 220 --> SPARE
   // SIGNAL 221 --> SPARE
   // SIGNAL 222 --> SPARE
   // SIGNAL 223 --> SPARE
   // SIGNAL 224 --> SPARE
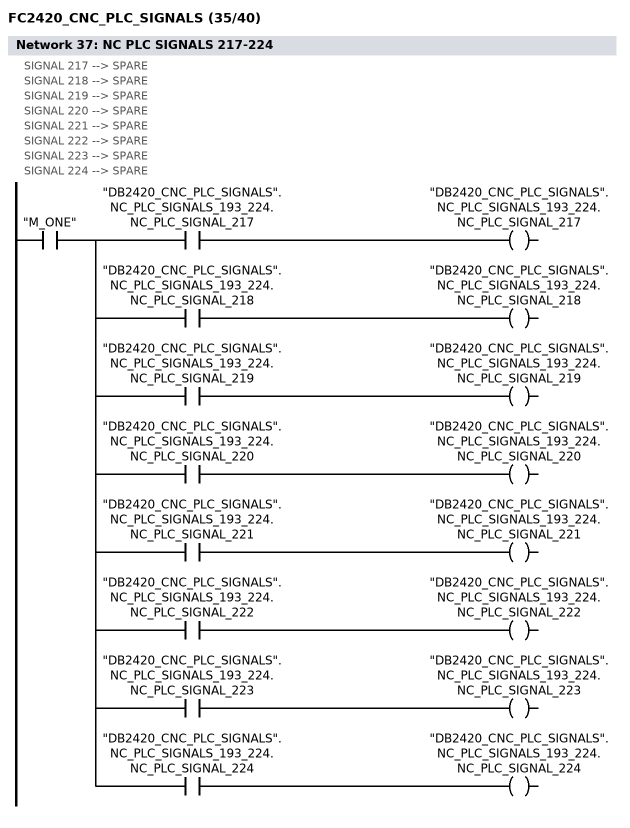
   RUNG wire#powerrail
      Contact( "M_ONE" )
      wire#w1
      Contact( "DB2420_CNC_PLC_SIGNALS".NC_PLC_SIGNALS_193_224.NC_PLC_SIGNAL_217 )
      Coil( "DB2420_CNC_PLC_SIGNALS".NC_PLC_SIGNALS_193_224.NC_PLC_SIGNAL_217 )
   END_RUNG
   RUNG wire#w1
      Contact( "DB2420_CNC_PLC_SIGNALS".NC_PLC_SIGNALS_193_224.NC_PLC_SIGNAL_218 )
      Coil( "DB2420_CNC_PLC_SIGNALS".NC_PLC_SIGNALS_193_224.NC_PLC_SIGNAL_218 )
   END_RUNG
   RUNG wire#w1
      Contact( "DB2420_CNC_PLC_SIGNALS".NC_PLC_SIGNALS_193_224.NC_PLC_SIGNAL_219 )
      Coil( "DB2420_CNC_PLC_SIGNALS".NC_PLC_SIGNALS_193_224.NC_PLC_SIGNAL_219 )
   END_RUNG
   RUNG wire#w1
      Contact( "DB2420_CNC_PLC_SIGNALS".NC_PLC_SIGNALS_193_224.NC_PLC_SIGNAL_220 )
      Coil( "DB2420_CNC_PLC_SIGNALS".NC_PLC_SIGNALS_193_224.NC_PLC_SIGNAL_220 )
   END_RUNG
   RUNG wire#w1
      Contact( "DB2420_CNC_PLC_SIGNALS".NC_PLC_SIGNALS_193_224.NC_PLC_SIGNAL_221 )
      Coil( "DB2420_CNC_PLC_SIGNALS".NC_PLC_SIGNALS_193_224.NC_PLC_SIGNAL_221 )
   END_RUNG
   RUNG wire#w1
      Contact( "DB2420_CNC_PLC_SIGNALS".NC_PLC_SIGNALS_193_224.NC_PLC_SIGNAL_222 )
      Coil( "DB2420_CNC_PLC_SIGNALS".NC_PLC_SIGNALS_193_224.NC_PLC_SIGNAL_222 )
   END_RUNG
   RUNG wire#w1
      Contact( "DB2420_CNC_PLC_SIGNALS".NC_PLC_SIGNALS_193_224.NC_PLC_SIGNAL_223 )
      Coil( "DB2420_CNC_PLC_SIGNALS".NC_PLC_SIGNALS_193_224.NC_PLC_SIGNAL_223 )
   END_RUNG
   RUNG wire#w1
      Contact( "DB2420_CNC_PLC_SIGNALS".NC_PLC_SIGNALS_193_224.NC_PLC_SIGNAL_224 )
      Coil( "DB2420_CNC_PLC_SIGNALS".NC_PLC_SIGNALS_193_224.NC_PLC_SIGNAL_224 )
   END_RUNG
   // the same network as SCL:
   "DB2420_CNC_PLC_SIGNALS".NC_PLC_SIGNALS_193_224.NC_PLC_SIGNAL_217 := "M_ONE" AND "DB2420_CNC_PLC_SIGNALS".NC_PLC_SIGNALS_193_224.NC_PLC_SIGNAL_217;
   "DB2420_CNC_PLC_SIGNALS".NC_PLC_SIGNALS_193_224.NC_PLC_SIGNAL_218 := "M_ONE" AND "DB2420_CNC_PLC_SIGNALS".NC_PLC_SIGNALS_193_224.NC_PLC_SIGNAL_218;
   "DB2420_CNC_PLC_SIGNALS".NC_PLC_SIGNALS_193_224.NC_PLC_SIGNAL_219 := "M_ONE" AND "DB2420_CNC_PLC_SIGNALS".NC_PLC_SIGNALS_193_224.NC_PLC_SIGNAL_219;
   "DB2420_CNC_PLC_SIGNALS".NC_PLC_SIGNALS_193_224.NC_PLC_SIGNAL_220 := "M_ONE" AND "DB2420_CNC_PLC_SIGNALS".NC_PLC_SIGNALS_193_224.NC_PLC_SIGNAL_220;
   "DB2420_CNC_PLC_SIGNALS".NC_PLC_SIGNALS_193_224.NC_PLC_SIGNAL_221 := "M_ONE" AND "DB2420_CNC_PLC_SIGNALS".NC_PLC_SIGNALS_193_224.NC_PLC_SIGNAL_221;
   "DB2420_CNC_PLC_SIGNALS".NC_PLC_SIGNALS_193_224.NC_PLC_SIGNAL_222 := "M_ONE" AND "DB2420_CNC_PLC_SIGNALS".NC_PLC_SIGNALS_193_224.NC_PLC_SIGNAL_222;
   "DB2420_CNC_PLC_SIGNALS".NC_PLC_SIGNALS_193_224.NC_PLC_SIGNAL_223 := "M_ONE" AND "DB2420_CNC_PLC_SIGNALS".NC_PLC_SIGNALS_193_224.NC_PLC_SIGNAL_223;
   "DB2420_CNC_PLC_SIGNALS".NC_PLC_SIGNALS_193_224.NC_PLC_SIGNAL_224 := "M_ONE" AND "DB2420_CNC_PLC_SIGNALS".NC_PLC_SIGNALS_193_224.NC_PLC_SIGNAL_224;
END_REGION

REGION Network 38: CALL FC21 NC PLC SIGNALS- $A_DBD[4068] / WRITE UNIT CYCLE SELECTION TO CNC
   // $A_DBD[1000] IN CNC
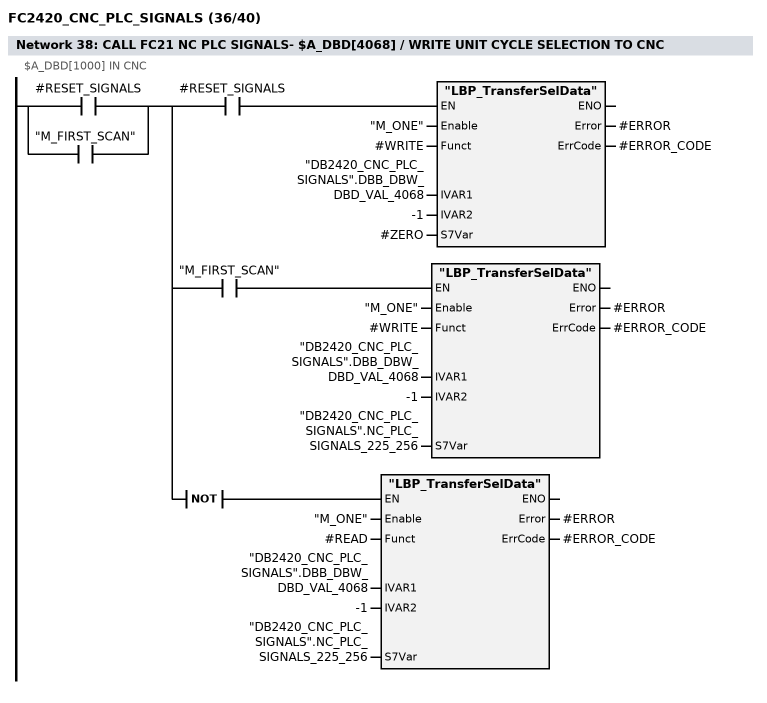
   RUNG wire#powerrail
      Contact( #RESET_SIGNALS )
      wire#w1
      Contact( #RESET_SIGNALS )
      "LBP_TransferSelData"(Enable := "M_ONE", Funct := #WRITE, IVAR1 := "DB2420_CNC_PLC_SIGNALS".DBB_DBW_DBD_VAL_4068, IVAR2 := -1, S7Var := #ZERO, Error => #ERROR, ErrCode => #ERROR_CODE)
   END_RUNG
   RUNG wire#powerrail
      Contact( "M_FIRST_SCAN" )
   END_RUNG wire#w1
   RUNG wire#w1
      Contact( "M_FIRST_SCAN" )
      "LBP_TransferSelData"(Enable := "M_ONE", Funct := #WRITE, IVAR1 := "DB2420_CNC_PLC_SIGNALS".DBB_DBW_DBD_VAL_4068, IVAR2 := -1, S7Var := "DB2420_CNC_PLC_SIGNALS".NC_PLC_SIGNALS_225_256, Error => #ERROR, ErrCode => #ERROR_CODE)
   END_RUNG
   RUNG wire#w1
      Not()
      "LBP_TransferSelData"(Enable := "M_ONE", Funct := #READ, IVAR1 := "DB2420_CNC_PLC_SIGNALS".DBB_DBW_DBD_VAL_4068, IVAR2 := -1, S7Var := "DB2420_CNC_PLC_SIGNALS".NC_PLC_SIGNALS_225_256, Error => #ERROR, ErrCode => #ERROR_CODE)
   END_RUNG
   // the same network as SCL:
   #_w1 := #RESET_SIGNALS OR "M_FIRST_SCAN";
   IF #_w1 AND #RESET_SIGNALS THEN
       "LBP_TransferSelData"(Enable := "M_ONE",
                             Funct := #WRITE,
                             IVAR1 := "DB2420_CNC_PLC_SIGNALS".DBB_DBW_DBD_VAL_4068,
                             IVAR2 := -1,
                             S7Var := #ZERO,
                             Error => #ERROR,
                             ErrCode => #ERROR_CODE);
   END_IF;
   IF #_w1 AND "M_FIRST_SCAN" THEN
       "LBP_TransferSelData"(Enable := "M_ONE",
                             Funct := #WRITE,
                             IVAR1 := "DB2420_CNC_PLC_SIGNALS".DBB_DBW_DBD_VAL_4068,
                             IVAR2 := -1,
                             S7Var := "DB2420_CNC_PLC_SIGNALS".NC_PLC_SIGNALS_225_256,
                             Error => #ERROR,
                             ErrCode => #ERROR_CODE);
   END_IF;
   IF NOT #_w1 THEN
       "LBP_TransferSelData"(Enable := "M_ONE",
                             Funct := #READ,
                             IVAR1 := "DB2420_CNC_PLC_SIGNALS".DBB_DBW_DBD_VAL_4068,
                             IVAR2 := -1,
                             S7Var := "DB2420_CNC_PLC_SIGNALS".NC_PLC_SIGNALS_225_256,
                             Error => #ERROR,
                             ErrCode => #ERROR_CODE);
   END_IF;
END_REGION

REGION Network 39: NC PLC SIGNALS 225-232
   // SIGNAL 225 --> SPARE
   // SIGNAL 226 --> SPARE
   // SIGNAL 227 --> SPARE
   // SIGNAL 228 --> SPARE
   // SIGNAL 229 --> SPARE
   // SIGNAL 230 --> SPARE
   // SIGNAL 231 --> SPARE
   // SIGNAL 232 --> SPARE
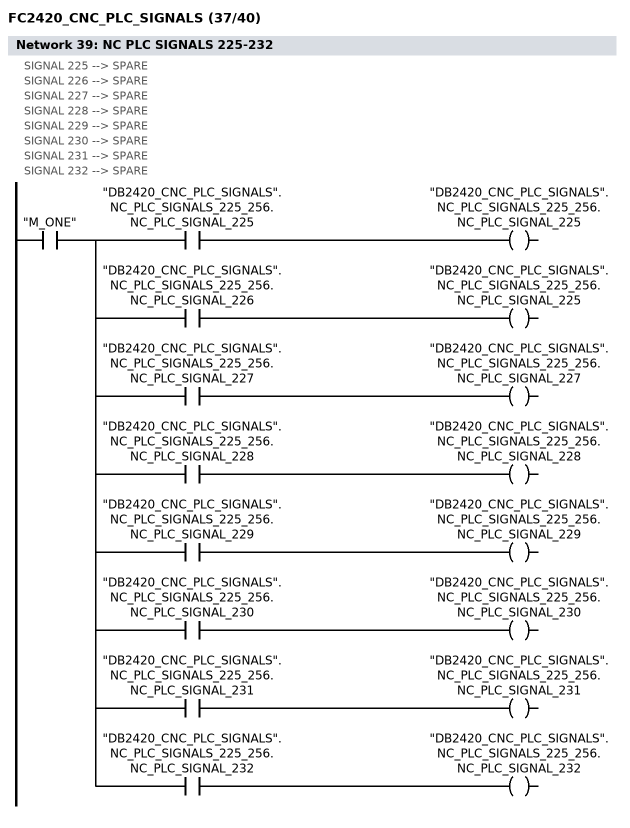
   RUNG wire#powerrail
      Contact( "M_ONE" )
      wire#w1
      Contact( "DB2420_CNC_PLC_SIGNALS".NC_PLC_SIGNALS_225_256.NC_PLC_SIGNAL_225 )
      Coil( "DB2420_CNC_PLC_SIGNALS".NC_PLC_SIGNALS_225_256.NC_PLC_SIGNAL_225 )
   END_RUNG
   RUNG wire#w1
      Contact( "DB2420_CNC_PLC_SIGNALS".NC_PLC_SIGNALS_225_256.NC_PLC_SIGNAL_226 )
      Coil( "DB2420_CNC_PLC_SIGNALS".NC_PLC_SIGNALS_225_256.NC_PLC_SIGNAL_225 )
   END_RUNG
   RUNG wire#w1
      Contact( "DB2420_CNC_PLC_SIGNALS".NC_PLC_SIGNALS_225_256.NC_PLC_SIGNAL_227 )
      Coil( "DB2420_CNC_PLC_SIGNALS".NC_PLC_SIGNALS_225_256.NC_PLC_SIGNAL_227 )
   END_RUNG
   RUNG wire#w1
      Contact( "DB2420_CNC_PLC_SIGNALS".NC_PLC_SIGNALS_225_256.NC_PLC_SIGNAL_228 )
      Coil( "DB2420_CNC_PLC_SIGNALS".NC_PLC_SIGNALS_225_256.NC_PLC_SIGNAL_228 )
   END_RUNG
   RUNG wire#w1
      Contact( "DB2420_CNC_PLC_SIGNALS".NC_PLC_SIGNALS_225_256.NC_PLC_SIGNAL_229 )
      Coil( "DB2420_CNC_PLC_SIGNALS".NC_PLC_SIGNALS_225_256.NC_PLC_SIGNAL_229 )
   END_RUNG
   RUNG wire#w1
      Contact( "DB2420_CNC_PLC_SIGNALS".NC_PLC_SIGNALS_225_256.NC_PLC_SIGNAL_230 )
      Coil( "DB2420_CNC_PLC_SIGNALS".NC_PLC_SIGNALS_225_256.NC_PLC_SIGNAL_230 )
   END_RUNG
   RUNG wire#w1
      Contact( "DB2420_CNC_PLC_SIGNALS".NC_PLC_SIGNALS_225_256.NC_PLC_SIGNAL_231 )
      Coil( "DB2420_CNC_PLC_SIGNALS".NC_PLC_SIGNALS_225_256.NC_PLC_SIGNAL_231 )
   END_RUNG
   RUNG wire#w1
      Contact( "DB2420_CNC_PLC_SIGNALS".NC_PLC_SIGNALS_225_256.NC_PLC_SIGNAL_232 )
      Coil( "DB2420_CNC_PLC_SIGNALS".NC_PLC_SIGNALS_225_256.NC_PLC_SIGNAL_232 )
   END_RUNG
   // the same network as SCL:
   "DB2420_CNC_PLC_SIGNALS".NC_PLC_SIGNALS_225_256.NC_PLC_SIGNAL_225 := "M_ONE" AND "DB2420_CNC_PLC_SIGNALS".NC_PLC_SIGNALS_225_256.NC_PLC_SIGNAL_225;
   "DB2420_CNC_PLC_SIGNALS".NC_PLC_SIGNALS_225_256.NC_PLC_SIGNAL_225 := "M_ONE" AND "DB2420_CNC_PLC_SIGNALS".NC_PLC_SIGNALS_225_256.NC_PLC_SIGNAL_226;
   "DB2420_CNC_PLC_SIGNALS".NC_PLC_SIGNALS_225_256.NC_PLC_SIGNAL_227 := "M_ONE" AND "DB2420_CNC_PLC_SIGNALS".NC_PLC_SIGNALS_225_256.NC_PLC_SIGNAL_227;
   "DB2420_CNC_PLC_SIGNALS".NC_PLC_SIGNALS_225_256.NC_PLC_SIGNAL_228 := "M_ONE" AND "DB2420_CNC_PLC_SIGNALS".NC_PLC_SIGNALS_225_256.NC_PLC_SIGNAL_228;
   "DB2420_CNC_PLC_SIGNALS".NC_PLC_SIGNALS_225_256.NC_PLC_SIGNAL_229 := "M_ONE" AND "DB2420_CNC_PLC_SIGNALS".NC_PLC_SIGNALS_225_256.NC_PLC_SIGNAL_229;
   "DB2420_CNC_PLC_SIGNALS".NC_PLC_SIGNALS_225_256.NC_PLC_SIGNAL_230 := "M_ONE" AND "DB2420_CNC_PLC_SIGNALS".NC_PLC_SIGNALS_225_256.NC_PLC_SIGNAL_230;
   "DB2420_CNC_PLC_SIGNALS".NC_PLC_SIGNALS_225_256.NC_PLC_SIGNAL_231 := "M_ONE" AND "DB2420_CNC_PLC_SIGNALS".NC_PLC_SIGNALS_225_256.NC_PLC_SIGNAL_231;
   "DB2420_CNC_PLC_SIGNALS".NC_PLC_SIGNALS_225_256.NC_PLC_SIGNAL_232 := "M_ONE" AND "DB2420_CNC_PLC_SIGNALS".NC_PLC_SIGNALS_225_256.NC_PLC_SIGNAL_232;
END_REGION

REGION Network 40: NC PLC SIGNALS 233-240
   // SIGNAL 233 --> SPARE
   // SIGNAL 234 --> SPARE
   // SIGNAL 235 --> SPARE
   // SIGNAL 236 --> SPARE
   // SIGNAL 237 --> SPARE
   // SIGNAL 238 --> SPARE
   // SIGNAL 239 --> SPARE
   // SIGNAL 240 --> SPARE
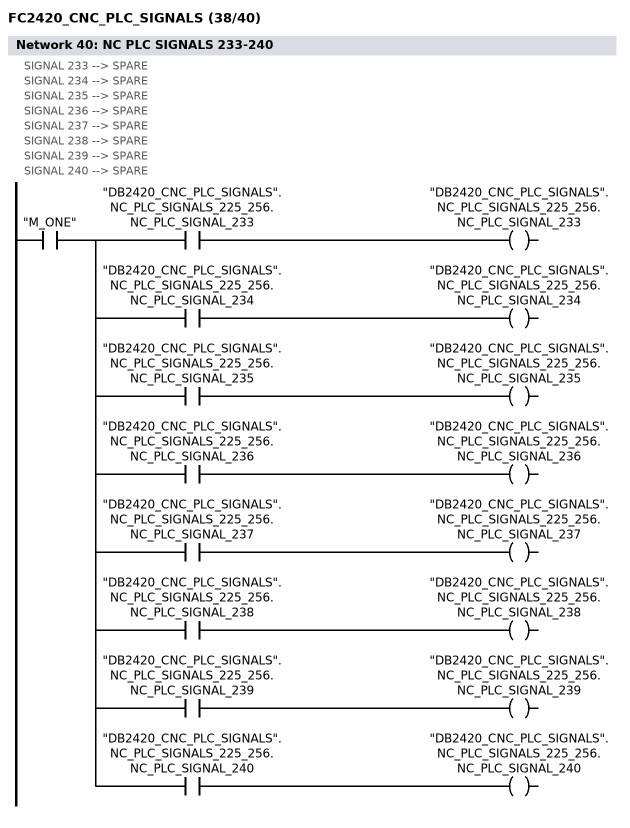
   RUNG wire#powerrail
      Contact( "M_ONE" )
      wire#w1
      Contact( "DB2420_CNC_PLC_SIGNALS".NC_PLC_SIGNALS_225_256.NC_PLC_SIGNAL_233 )
      Coil( "DB2420_CNC_PLC_SIGNALS".NC_PLC_SIGNALS_225_256.NC_PLC_SIGNAL_233 )
   END_RUNG
   RUNG wire#w1
      Contact( "DB2420_CNC_PLC_SIGNALS".NC_PLC_SIGNALS_225_256.NC_PLC_SIGNAL_234 )
      Coil( "DB2420_CNC_PLC_SIGNALS".NC_PLC_SIGNALS_225_256.NC_PLC_SIGNAL_234 )
   END_RUNG
   RUNG wire#w1
      Contact( "DB2420_CNC_PLC_SIGNALS".NC_PLC_SIGNALS_225_256.NC_PLC_SIGNAL_235 )
      Coil( "DB2420_CNC_PLC_SIGNALS".NC_PLC_SIGNALS_225_256.NC_PLC_SIGNAL_235 )
   END_RUNG
   RUNG wire#w1
      Contact( "DB2420_CNC_PLC_SIGNALS".NC_PLC_SIGNALS_225_256.NC_PLC_SIGNAL_236 )
      Coil( "DB2420_CNC_PLC_SIGNALS".NC_PLC_SIGNALS_225_256.NC_PLC_SIGNAL_236 )
   END_RUNG
   RUNG wire#w1
      Contact( "DB2420_CNC_PLC_SIGNALS".NC_PLC_SIGNALS_225_256.NC_PLC_SIGNAL_237 )
      Coil( "DB2420_CNC_PLC_SIGNALS".NC_PLC_SIGNALS_225_256.NC_PLC_SIGNAL_237 )
   END_RUNG
   RUNG wire#w1
      Contact( "DB2420_CNC_PLC_SIGNALS".NC_PLC_SIGNALS_225_256.NC_PLC_SIGNAL_238 )
      Coil( "DB2420_CNC_PLC_SIGNALS".NC_PLC_SIGNALS_225_256.NC_PLC_SIGNAL_238 )
   END_RUNG
   RUNG wire#w1
      Contact( "DB2420_CNC_PLC_SIGNALS".NC_PLC_SIGNALS_225_256.NC_PLC_SIGNAL_239 )
      Coil( "DB2420_CNC_PLC_SIGNALS".NC_PLC_SIGNALS_225_256.NC_PLC_SIGNAL_239 )
   END_RUNG
   RUNG wire#w1
      Contact( "DB2420_CNC_PLC_SIGNALS".NC_PLC_SIGNALS_225_256.NC_PLC_SIGNAL_240 )
      Coil( "DB2420_CNC_PLC_SIGNALS".NC_PLC_SIGNALS_225_256.NC_PLC_SIGNAL_240 )
   END_RUNG
   // the same network as SCL:
   "DB2420_CNC_PLC_SIGNALS".NC_PLC_SIGNALS_225_256.NC_PLC_SIGNAL_233 := "M_ONE" AND "DB2420_CNC_PLC_SIGNALS".NC_PLC_SIGNALS_225_256.NC_PLC_SIGNAL_233;
   "DB2420_CNC_PLC_SIGNALS".NC_PLC_SIGNALS_225_256.NC_PLC_SIGNAL_234 := "M_ONE" AND "DB2420_CNC_PLC_SIGNALS".NC_PLC_SIGNALS_225_256.NC_PLC_SIGNAL_234;
   "DB2420_CNC_PLC_SIGNALS".NC_PLC_SIGNALS_225_256.NC_PLC_SIGNAL_235 := "M_ONE" AND "DB2420_CNC_PLC_SIGNALS".NC_PLC_SIGNALS_225_256.NC_PLC_SIGNAL_235;
   "DB2420_CNC_PLC_SIGNALS".NC_PLC_SIGNALS_225_256.NC_PLC_SIGNAL_236 := "M_ONE" AND "DB2420_CNC_PLC_SIGNALS".NC_PLC_SIGNALS_225_256.NC_PLC_SIGNAL_236;
   "DB2420_CNC_PLC_SIGNALS".NC_PLC_SIGNALS_225_256.NC_PLC_SIGNAL_237 := "M_ONE" AND "DB2420_CNC_PLC_SIGNALS".NC_PLC_SIGNALS_225_256.NC_PLC_SIGNAL_237;
   "DB2420_CNC_PLC_SIGNALS".NC_PLC_SIGNALS_225_256.NC_PLC_SIGNAL_238 := "M_ONE" AND "DB2420_CNC_PLC_SIGNALS".NC_PLC_SIGNALS_225_256.NC_PLC_SIGNAL_238;
   "DB2420_CNC_PLC_SIGNALS".NC_PLC_SIGNALS_225_256.NC_PLC_SIGNAL_239 := "M_ONE" AND "DB2420_CNC_PLC_SIGNALS".NC_PLC_SIGNALS_225_256.NC_PLC_SIGNAL_239;
   "DB2420_CNC_PLC_SIGNALS".NC_PLC_SIGNALS_225_256.NC_PLC_SIGNAL_240 := "M_ONE" AND "DB2420_CNC_PLC_SIGNALS".NC_PLC_SIGNALS_225_256.NC_PLC_SIGNAL_240;
END_REGION

REGION Network 41: NC PLC SIGNALS 241-248
   // SIGNAL 241 --> SPARE
   // SIGNAL 242 --> SPARE
   // SIGNAL 243 --> SPARE
   // SIGNAL 244 --> SPARE
   // SIGNAL 245 --> SPARE
   // SIGNAL 246 --> SPARE
   // SIGNAL 247 --> SPARE
   // SIGNAL 248 --> SPARE
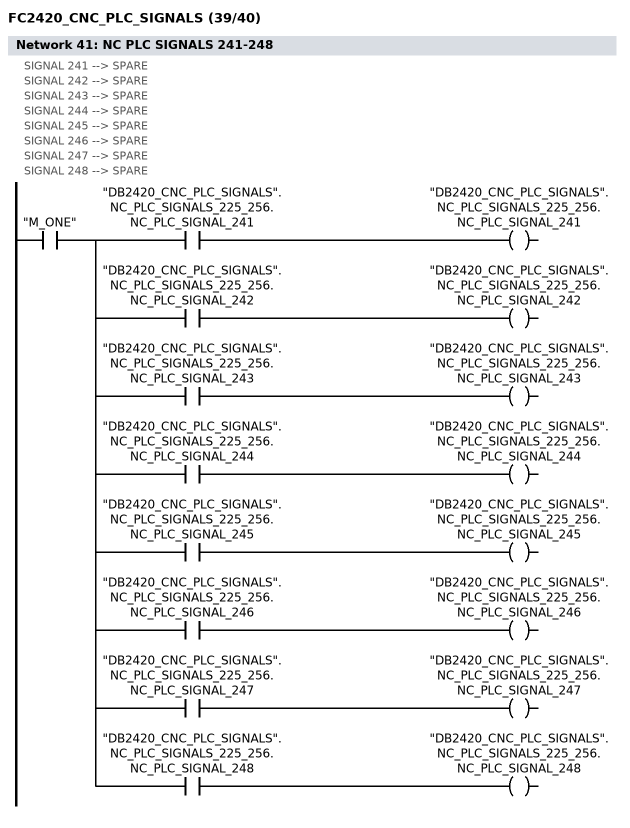
   RUNG wire#powerrail
      Contact( "M_ONE" )
      wire#w1
      Contact( "DB2420_CNC_PLC_SIGNALS".NC_PLC_SIGNALS_225_256.NC_PLC_SIGNAL_241 )
      Coil( "DB2420_CNC_PLC_SIGNALS".NC_PLC_SIGNALS_225_256.NC_PLC_SIGNAL_241 )
   END_RUNG
   RUNG wire#w1
      Contact( "DB2420_CNC_PLC_SIGNALS".NC_PLC_SIGNALS_225_256.NC_PLC_SIGNAL_242 )
      Coil( "DB2420_CNC_PLC_SIGNALS".NC_PLC_SIGNALS_225_256.NC_PLC_SIGNAL_242 )
   END_RUNG
   RUNG wire#w1
      Contact( "DB2420_CNC_PLC_SIGNALS".NC_PLC_SIGNALS_225_256.NC_PLC_SIGNAL_243 )
      Coil( "DB2420_CNC_PLC_SIGNALS".NC_PLC_SIGNALS_225_256.NC_PLC_SIGNAL_243 )
   END_RUNG
   RUNG wire#w1
      Contact( "DB2420_CNC_PLC_SIGNALS".NC_PLC_SIGNALS_225_256.NC_PLC_SIGNAL_244 )
      Coil( "DB2420_CNC_PLC_SIGNALS".NC_PLC_SIGNALS_225_256.NC_PLC_SIGNAL_244 )
   END_RUNG
   RUNG wire#w1
      Contact( "DB2420_CNC_PLC_SIGNALS".NC_PLC_SIGNALS_225_256.NC_PLC_SIGNAL_245 )
      Coil( "DB2420_CNC_PLC_SIGNALS".NC_PLC_SIGNALS_225_256.NC_PLC_SIGNAL_245 )
   END_RUNG
   RUNG wire#w1
      Contact( "DB2420_CNC_PLC_SIGNALS".NC_PLC_SIGNALS_225_256.NC_PLC_SIGNAL_246 )
      Coil( "DB2420_CNC_PLC_SIGNALS".NC_PLC_SIGNALS_225_256.NC_PLC_SIGNAL_246 )
   END_RUNG
   RUNG wire#w1
      Contact( "DB2420_CNC_PLC_SIGNALS".NC_PLC_SIGNALS_225_256.NC_PLC_SIGNAL_247 )
      Coil( "DB2420_CNC_PLC_SIGNALS".NC_PLC_SIGNALS_225_256.NC_PLC_SIGNAL_247 )
   END_RUNG
   RUNG wire#w1
      Contact( "DB2420_CNC_PLC_SIGNALS".NC_PLC_SIGNALS_225_256.NC_PLC_SIGNAL_248 )
      Coil( "DB2420_CNC_PLC_SIGNALS".NC_PLC_SIGNALS_225_256.NC_PLC_SIGNAL_248 )
   END_RUNG
   // the same network as SCL:
   "DB2420_CNC_PLC_SIGNALS".NC_PLC_SIGNALS_225_256.NC_PLC_SIGNAL_241 := "M_ONE" AND "DB2420_CNC_PLC_SIGNALS".NC_PLC_SIGNALS_225_256.NC_PLC_SIGNAL_241;
   "DB2420_CNC_PLC_SIGNALS".NC_PLC_SIGNALS_225_256.NC_PLC_SIGNAL_242 := "M_ONE" AND "DB2420_CNC_PLC_SIGNALS".NC_PLC_SIGNALS_225_256.NC_PLC_SIGNAL_242;
   "DB2420_CNC_PLC_SIGNALS".NC_PLC_SIGNALS_225_256.NC_PLC_SIGNAL_243 := "M_ONE" AND "DB2420_CNC_PLC_SIGNALS".NC_PLC_SIGNALS_225_256.NC_PLC_SIGNAL_243;
   "DB2420_CNC_PLC_SIGNALS".NC_PLC_SIGNALS_225_256.NC_PLC_SIGNAL_244 := "M_ONE" AND "DB2420_CNC_PLC_SIGNALS".NC_PLC_SIGNALS_225_256.NC_PLC_SIGNAL_244;
   "DB2420_CNC_PLC_SIGNALS".NC_PLC_SIGNALS_225_256.NC_PLC_SIGNAL_245 := "M_ONE" AND "DB2420_CNC_PLC_SIGNALS".NC_PLC_SIGNALS_225_256.NC_PLC_SIGNAL_245;
   "DB2420_CNC_PLC_SIGNALS".NC_PLC_SIGNALS_225_256.NC_PLC_SIGNAL_246 := "M_ONE" AND "DB2420_CNC_PLC_SIGNALS".NC_PLC_SIGNALS_225_256.NC_PLC_SIGNAL_246;
   "DB2420_CNC_PLC_SIGNALS".NC_PLC_SIGNALS_225_256.NC_PLC_SIGNAL_247 := "M_ONE" AND "DB2420_CNC_PLC_SIGNALS".NC_PLC_SIGNALS_225_256.NC_PLC_SIGNAL_247;
   "DB2420_CNC_PLC_SIGNALS".NC_PLC_SIGNALS_225_256.NC_PLC_SIGNAL_248 := "M_ONE" AND "DB2420_CNC_PLC_SIGNALS".NC_PLC_SIGNALS_225_256.NC_PLC_SIGNAL_248;
END_REGION

REGION Network 42: NC PLC SIGNALS 249-256
   // SIGNAL 249 --> SPARE
   // SIGNAL 250 --> SPARE
   // SIGNAL 251 --> SPARE
   // SIGNAL 252 --> SPARE
   // SIGNAL 253 --> SPARE
   // SIGNAL 254 --> SPARE
   // SIGNAL 255 --> SPARE
   // SIGNAL 256 --> SPARE
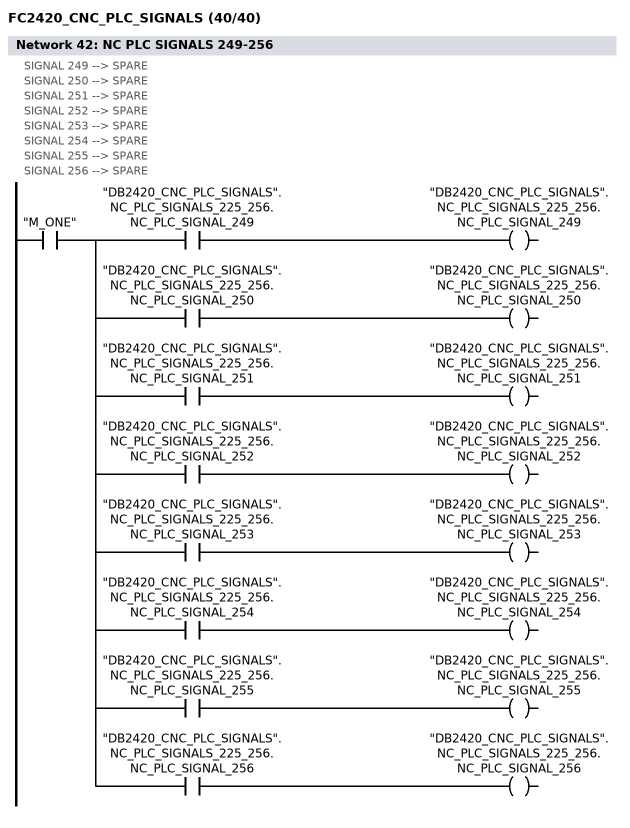
   RUNG wire#powerrail
      Contact( "M_ONE" )
      wire#w1
      Contact( "DB2420_CNC_PLC_SIGNALS".NC_PLC_SIGNALS_225_256.NC_PLC_SIGNAL_249 )
      Coil( "DB2420_CNC_PLC_SIGNALS".NC_PLC_SIGNALS_225_256.NC_PLC_SIGNAL_249 )
   END_RUNG
   RUNG wire#w1
      Contact( "DB2420_CNC_PLC_SIGNALS".NC_PLC_SIGNALS_225_256.NC_PLC_SIGNAL_250 )
      Coil( "DB2420_CNC_PLC_SIGNALS".NC_PLC_SIGNALS_225_256.NC_PLC_SIGNAL_250 )
   END_RUNG
   RUNG wire#w1
      Contact( "DB2420_CNC_PLC_SIGNALS".NC_PLC_SIGNALS_225_256.NC_PLC_SIGNAL_251 )
      Coil( "DB2420_CNC_PLC_SIGNALS".NC_PLC_SIGNALS_225_256.NC_PLC_SIGNAL_251 )
   END_RUNG
   RUNG wire#w1
      Contact( "DB2420_CNC_PLC_SIGNALS".NC_PLC_SIGNALS_225_256.NC_PLC_SIGNAL_252 )
      Coil( "DB2420_CNC_PLC_SIGNALS".NC_PLC_SIGNALS_225_256.NC_PLC_SIGNAL_252 )
   END_RUNG
   RUNG wire#w1
      Contact( "DB2420_CNC_PLC_SIGNALS".NC_PLC_SIGNALS_225_256.NC_PLC_SIGNAL_253 )
      Coil( "DB2420_CNC_PLC_SIGNALS".NC_PLC_SIGNALS_225_256.NC_PLC_SIGNAL_253 )
   END_RUNG
   RUNG wire#w1
      Contact( "DB2420_CNC_PLC_SIGNALS".NC_PLC_SIGNALS_225_256.NC_PLC_SIGNAL_254 )
      Coil( "DB2420_CNC_PLC_SIGNALS".NC_PLC_SIGNALS_225_256.NC_PLC_SIGNAL_254 )
   END_RUNG
   RUNG wire#w1
      Contact( "DB2420_CNC_PLC_SIGNALS".NC_PLC_SIGNALS_225_256.NC_PLC_SIGNAL_255 )
      Coil( "DB2420_CNC_PLC_SIGNALS".NC_PLC_SIGNALS_225_256.NC_PLC_SIGNAL_255 )
   END_RUNG
   RUNG wire#w1
      Contact( "DB2420_CNC_PLC_SIGNALS".NC_PLC_SIGNALS_225_256.NC_PLC_SIGNAL_256 )
      Coil( "DB2420_CNC_PLC_SIGNALS".NC_PLC_SIGNALS_225_256.NC_PLC_SIGNAL_256 )
   END_RUNG
   // the same network as SCL:
   "DB2420_CNC_PLC_SIGNALS".NC_PLC_SIGNALS_225_256.NC_PLC_SIGNAL_249 := "M_ONE" AND "DB2420_CNC_PLC_SIGNALS".NC_PLC_SIGNALS_225_256.NC_PLC_SIGNAL_249;
   "DB2420_CNC_PLC_SIGNALS".NC_PLC_SIGNALS_225_256.NC_PLC_SIGNAL_250 := "M_ONE" AND "DB2420_CNC_PLC_SIGNALS".NC_PLC_SIGNALS_225_256.NC_PLC_SIGNAL_250;
   "DB2420_CNC_PLC_SIGNALS".NC_PLC_SIGNALS_225_256.NC_PLC_SIGNAL_251 := "M_ONE" AND "DB2420_CNC_PLC_SIGNALS".NC_PLC_SIGNALS_225_256.NC_PLC_SIGNAL_251;
   "DB2420_CNC_PLC_SIGNALS".NC_PLC_SIGNALS_225_256.NC_PLC_SIGNAL_252 := "M_ONE" AND "DB2420_CNC_PLC_SIGNALS".NC_PLC_SIGNALS_225_256.NC_PLC_SIGNAL_252;
   "DB2420_CNC_PLC_SIGNALS".NC_PLC_SIGNALS_225_256.NC_PLC_SIGNAL_253 := "M_ONE" AND "DB2420_CNC_PLC_SIGNALS".NC_PLC_SIGNALS_225_256.NC_PLC_SIGNAL_253;
   "DB2420_CNC_PLC_SIGNALS".NC_PLC_SIGNALS_225_256.NC_PLC_SIGNAL_254 := "M_ONE" AND "DB2420_CNC_PLC_SIGNALS".NC_PLC_SIGNALS_225_256.NC_PLC_SIGNAL_254;
   "DB2420_CNC_PLC_SIGNALS".NC_PLC_SIGNALS_225_256.NC_PLC_SIGNAL_255 := "M_ONE" AND "DB2420_CNC_PLC_SIGNALS".NC_PLC_SIGNALS_225_256.NC_PLC_SIGNAL_255;
   "DB2420_CNC_PLC_SIGNALS".NC_PLC_SIGNALS_225_256.NC_PLC_SIGNAL_256 := "M_ONE" AND "DB2420_CNC_PLC_SIGNALS".NC_PLC_SIGNALS_225_256.NC_PLC_SIGNAL_256;
END_REGION
END_FUNCTION
